// TIA Portal V18 program export: 1 tag tables, 1 data types, 57 data blocks, 50 code blocks (in call order from the OBs), 135 instance data blocks

VAR_GLOBAL   // PLC tag table "Default tag table"
   "Alarm Drive1" AT %I0.0 : Bool;
   "Alarm Drive 2" AT %I0.1 : Bool;
   setFlowRate AT %IW64 : Int;
   "AI on board(1)" AT %IW102 : Int;
   "preliminary empty signal component B1" AT %I0.6 : Bool;
   "Metering Start Foot Switch" AT %I1.2 : Bool;
   "Metering Start" AT %I1.3 : Bool;
   "Metering Stop" AT %I1.4 : Bool;
   "Metering Function Selection" AT %I2.0 : Bool;
   "Prerun Function" AT %I2.1 : Bool;
   "level empty signal component B1" AT %I0.7 : Bool;
   Flush AT %I2.2 : Bool;
   "Pressure sensor Pump Inlet A" AT %IW112 : Int;
   "Pressure Sensor Pump Inlet B" AT %IW114 : Int;
   "Pressure Sensor Pump Outlet A" AT %IW116 : Int;
   "Pressure Sensor Pump Outlet B" AT %IW118 : Int;
   "RPM PUMP A" AT %ID1008 : DInt;
   "RPM PUMP B" AT %ID1012 : DInt;
   "Level empty Signal component A1" AT %I0.3 : Bool;
   "program selection bit 3" AT %I2.6 : Bool;
   "preliminary empty signal component A1" AT %I0.2 : Bool;
   "Program selection bit0" AT %I2.3 : Bool;   //    {ExternalWritable false}
   "program selection bit 1" AT %I2.4 : Bool;
   "program selection bit2" AT %I2.5 : Bool;
   "Regenration Position Reached" AT %I1.5 : Bool;
   "reset pb" AT %I2.7 : Bool;
   "preliminary empty signal component A2" AT %I0.4 : Bool;
   "Level empty Signal component A2" AT %I0.5 : Bool;
   "preliminary empty signal component B2" AT %I1.0 : Bool;
   "level empty signal component B2" AT %I1.1 : Bool;
   "Level Sensor A" AT %IW120 : Int;
   "Level Sensor B" AT %IW122 : Int;
   "Pressure sensor Pump Inlet A_mA" AT %IW124 : Int;
   "Pressure Sensor Pump Inlet B_mA" AT %IW126 : Int;
   "emergency stop" AT %M3.5 : Bool;
   heater1 AT %IW144 : Int;
   heater2 AT %IW146 : Int;
   heater3 AT %IW148 : Int;
   heater4 AT %IW150 : Int;
   "Control ON" AT %I3.0 : Bool;
   "Control ON Led" AT %Q1.0 : Bool;
   "Reserve out3" AT %Q1.1 : Bool;
   "Metering Running" AT %Q2.2 : Bool;
   "ready to meter" AT %Q2.0 : Bool;
   "Metering Fault" AT %Q2.5 : Bool;
   "General Alarm" AT %Q2.1 : Bool;
   "Waiting for pre run" AT %Q2.3 : Bool;
   "metering Completed" AT %Q2.4 : Bool;
   "tower lamp yellow" AT %Q0.5 : Bool;
   "Reserve out0" AT %Q0.6 : Bool;
   "Reserve out1" AT %Q0.7 : Bool;
   "potlife error" AT %Q2.6 : Bool;
   "Reserve Output6" AT %Q2.7 : Bool;
   buzzer AT %Q0.4 : Bool;
   "Gear Pump A On_FWD" AT %Q0.0 : Bool;
   "Gear Pump B On_FWD" AT %Q0.2 : Bool;
   speedReference_ComponentB AT %QW130 : Int;
   speedReference_ComponentA AT %QW128 : Int;
   rampReference_ComponentA AT %QW132 : Int;
   rampReference_ComponentB AT %QW134 : Int;
   "Gear Pump A On_REW" AT %Q0.1 : Bool;
   "Gear Pump B On_REW" AT %Q0.3 : Bool;
   "Material 1 Temperature output" AT %Q3.0 : Bool;
   "Material 2 Temperature output" AT %Q3.1 : Bool;
   "Material 3 Temperature output" AT %Q3.2 : Bool;
   "Material 4 Temperature output" AT %Q3.3 : Bool;
   "gear Pump A fault" AT %M100.1 : Bool;
   "gear Pump B fault" AT %M100.2 : Bool;
   "Outlet Component A On" AT %M261.4 : Bool;
   "Outlet Component B On" AT %M200.4 : Bool;
   "program selection bit4" AT %M100.5 : Bool;
   "Agitator B Fault" AT %M100.3 : Bool;
   "Phase sequence relay Failure" AT %M100.4 : Bool;
   "Part Present sensor" AT %M100.0 : Bool;
   "Metering Ready" AT %M201.2 : Bool;
   "Tank A1 pressure" AT %MW240 : Int;
   "Tank A2 pressure" AT %MW242 : Int;
   "Tank B1 pressure" AT %MW244 : Int;
   "Tank Level A2" AT %MW248 : Int;
   "Gear Pump A Speed" AT %MW128 : Int;
   "Gear Pump B Speed" AT %MW130 : Int;
   "Mixer Speed" AT %MW208 : Int;
   "reserve  Analog output_0" AT %MW210 : Int;
   System_Byte AT %MB1 : Byte;
   FirstScan AT %M1.0 : Bool;
   DiagStatusUpdate AT %M1.1 : Bool;
   AlwaysTRUE AT %M1.2 : Bool;
   AlwaysFALSE AT %M1.3 : Bool;
   Clock_Byte AT %MB0 : Byte;
   Clock_10Hz AT %M0.0 : Bool;
   Clock_5Hz AT %M0.1 : Bool;
   "Clock_2.5Hz" AT %M0.2 : Bool;
   Clock_2Hz AT %M0.3 : Bool;
   "Clock_1.25Hz" AT %M0.4 : Bool;
   Clock_1Hz AT %M0.5 : Bool;
   "Clock_0.625Hz" AT %M0.6 : Bool;
   "Clock_0.5Hz" AT %M0.7 : Bool;
   "Fault register 1" AT %MW60 : Word;
   "Fault register 2" AT %MW62 : Word;
   "Fault register 3" AT %MW64 : Word;
   "Fault register 4" AT %MW66 : Word;
   "Fault register 5" AT %MW68 : Word;
   "A1-emergency stop active" AT %M61.0 : Bool;
   "A2-Pump A Drive Fault" AT %M61.1 : Bool;
   "A3-pump B drive Fault" AT %M61.2 : Bool;
   "A4-Agitator A1 fault" AT %M61.3 : Bool;
   "A5-Agitator A2 fault" AT %M61.4 : Bool;
   "A6-Tank A level sensor fault" AT %M61.5 : Bool;
   "A7-Tank B level sensor fault" AT %M61.6 : Bool;
   "A8-Pump A pressure sensor fault" AT %M61.7 : Bool;
   "A9-Pump B pressure sensor fault" AT %M60.0 : Bool;
   "A10-Tank A1 level sensor fault" AT %M60.1 : Bool;
   "A11-Tank A Filling Error" AT %M60.2 : Bool;
   "A12-Heater1 sensor fault" AT %M60.3 : Bool;
   "A13-Heater2 sensor fault" AT %M60.4 : Bool;
   "A14-Heater3 sensor fault" AT %M60.5 : Bool;
   "A15-Heater4 sensor fault" AT %M60.6 : Bool;
   "A16-Vaccum pump A fault" AT %M60.7 : Bool;
   "A17-Heater1 undertemperature" AT %M63.0 : Bool;
   "A18-Heater2 undertemperature" AT %M63.1 : Bool;
   "A19-Heater3 undertemperature" AT %M63.2 : Bool;
   "A20-Heater4 undertemperature" AT %M63.3 : Bool;
   "A21- Heater1 overtemperature" AT %M63.4 : Bool;
   "A22- Heater2 overtemperature" AT %M63.5 : Bool;
   "A23- Heater3 overtemperature" AT %M63.6 : Bool;
   "A24- Heater4 overtemperature" AT %M63.7 : Bool;
   "A25- Heater 8 pt100 discooneted" AT %M62.0 : Bool;
   "A26- Heater 9 pt100 discooneted" AT %M62.1 : Bool;
   "A27- Heater 10 pt100 discooneted" AT %M62.2 : Bool;
   "A28- Pump A over pressure" AT %M62.3 : Bool;
   "A29-pump B Over pressure" AT %M62.4 : Bool;
   "A30-Tank A1 Level Empty" AT %M62.5 : Bool;
   "A31-Tank A2 Level Empty" AT %M62.6 : Bool;
   "A32-Tank B Level Empty" AT %M62.7 : Bool;
   "A33-Tank A1 low level" AT %M65.0 : Bool;
   "A34-Tank A2 low level" AT %M65.1 : Bool;
   "A35-Tank B low level" AT %M65.2 : Bool;
   "A36-Pump A lower pressure" AT %M65.3 : Bool;
   "A37-Pump B lower pressure" AT %M65.4 : Bool;
   "A38-A material Supply fault" AT %M65.5 : Bool;
   "A39-B material Supply fault" AT %M65.6 : Bool;
   "A40-Potlife elapsed Change static mixer" AT %M65.7 : Bool;
   "A41- Heater 1 temperature Low" AT %M64.0 : Bool;
   "A42- Heater 2 temperature Low" AT %M64.1 : Bool;
   "A43- Heater 3 temperature Low" AT %M64.2 : Bool;
   "A44- Heater 4 temperature Low" AT %M64.3 : Bool;
   "A45- Heater 5 temperature Low" AT %M64.4 : Bool;
   "A46- Heater 6 temperature Low" AT %M64.5 : Bool;
   "A47- Heater 7 temperature Low" AT %M64.6 : Bool;
   "A48- Heater 8 temperature Low" AT %M64.7 : Bool;
   "A49- heater 9 temperature low" AT %M67.0 : Bool;
   "A50- heater 10 temperature low" AT %M67.1 : Bool;
   "A51- heater 1 temperature high" AT %M67.2 : Bool;
   "A52- heater 2 temperature high" AT %M67.3 : Bool;
   "A53- heater 3 temperature high" AT %M67.4 : Bool;
   "A54- heater 4 temperature high" AT %M67.5 : Bool;
   "A55- heater 5 temperature high" AT %M67.6 : Bool;
   "A56- heater 6 temperature high" AT %M67.7 : Bool;
   "A57- heater  7 temperature high" AT %M66.0 : Bool;
   "A58- heater 8 temperature high" AT %M66.1 : Bool;
   "A59- heater 9 temperature high" AT %M66.2 : Bool;
   "A60- heater 10 temperature high" AT %M66.3 : Bool;
   "A61- refilling failed Tank A1" AT %M66.4 : Bool;
   "A62-Error flowrate" AT %M66.5 : Bool;
   "A63- refilling failed Tank B" AT %M66.6 : Bool;
   Ack_A1 AT %M341.0 : Bool;
   Ack_A2 AT %M341.1 : Bool;
   Ack_A3 AT %M341.2 : Bool;
   Ack_A4 AT %M341.3 : Bool;
   Ack_A5 AT %M341.4 : Bool;
   Ack_A6 AT %M341.5 : Bool;
   Ack_A7 AT %M341.6 : Bool;
   Ack_A8 AT %M341.7 : Bool;
   Ack_A9 AT %M342.0 : Bool;
   Ack_A10 AT %M342.1 : Bool;
   Ack_A11 AT %M342.2 : Bool;
   Ack_A12 AT %M342.3 : Bool;
   Ack_A13 AT %M342.4 : Bool;
   Ack_A14 AT %M342.5 : Bool;
   Ack_A15 AT %M342.6 : Bool;
   Ack_A16 AT %M342.7 : Bool;
   Ack_A17 AT %M343.0 : Bool;
   Ack_A18 AT %M343.1 : Bool;
   Ack_A19 AT %M343.2 : Bool;
   Ack_A20 AT %M343.3 : Bool;
   Ack_A21 AT %M343.4 : Bool;
   Ack_A22 AT %M343.5 : Bool;
   Ack_A23 AT %M343.6 : Bool;
   Ack_A24 AT %M343.7 : Bool;
   Ack_A25 AT %M344.0 : Bool;
   Ack_A26 AT %M344.1 : Bool;
   Ack_A27 AT %M344.2 : Bool;
   Ack_A28 AT %M344.3 : Bool;
   Ack_A29 AT %M344.4 : Bool;
   Ack_A30 AT %M344.5 : Bool;
   Ack_A31 AT %M344.6 : Bool;
   Ack_A32 AT %M344.7 : Bool;
   Ack_A33 AT %M345.0 : Bool;
   Ack_A34 AT %M345.1 : Bool;
   Ack_A35 AT %M345.2 : Bool;
   Ack_A36 AT %M345.3 : Bool;
   Ack_A37 AT %M345.4 : Bool;
   Ack_A38 AT %M345.5 : Bool;
   Ack_A39 AT %M345.6 : Bool;
   Ack_A40 AT %M345.7 : Bool;
   Ack_A41 AT %M346.0 : Bool;
   Ack_A42 AT %M346.1 : Bool;
   Ack_A43 AT %M346.2 : Bool;
   Ack_A44 AT %M346.3 : Bool;
   Ack_A45 AT %M346.4 : Bool;
   Ack_A46 AT %M346.5 : Bool;
   Ack_A47 AT %M346.6 : Bool;
   Ack_A48 AT %M346.7 : Bool;
   Ack_A49 AT %M347.0 : Bool;
   Ack_A50 AT %M347.1 : Bool;
   Ack_A51 AT %M347.2 : Bool;
   Ack_A52 AT %M347.3 : Bool;
   Ack_A53 AT %M347.4 : Bool;
   Ack_A54 AT %M347.5 : Bool;
   Ack_A55 AT %M347.6 : Bool;
   Ack_A56 AT %M347.7 : Bool;
   Ack_A57 AT %M348.0 : Bool;
   Ack_A58 AT %M348.1 : Bool;
   Ack_A59 AT %M348.2 : Bool;
   Ack_A60 AT %M348.3 : Bool;
   Ack_A61 AT %M348.4 : Bool;
   Ack_A62 AT %M348.5 : Bool;
   Ack_A63 AT %M348.6 : Bool;
   Ack_A64 AT %M348.7 : Bool;
   Ack_A65 AT %M349.0 : Bool;
   Ack_A66 AT %M349.1 : Bool;
   Ack_A67 AT %M349.2 : Bool;
   Ack_A68 AT %M349.3 : Bool;
   Ack_A69 AT %M349.4 : Bool;
   Ack_hmi AT %M39.0 : Bool;
   Ack_site AT %M39.1 : Bool;
   Ack_PB AT %M39.2 : Bool;
   Fault_Ack_ONS AT %M39.3 : Bool;
   Tag_1 AT %M21.0 : Bool;
   Tag_2 AT %M4.1 : Bool;
   Ack_hmi_ons AT %M39.4 : Bool;
   "1sec_pulse" AT %M2.0 : Bool;
   "transperant backround" AT %M5.0 : Bool;
   "error count" AT %MD6 : UDInt;
   "A66-Tank A1 over pressure" AT %M69.1 : Bool;
   "A67-Tank A2 over pressure" AT %M69.2 : Bool;
   "A68-Tank B1 over pressure" AT %M69.3 : Bool;
   "Pgm No site" AT %MW23 : Int;
   "Pgm selection Bit memory 1" AT %M23.0 : Bool;
   "Pgm selection Bit memory 2" AT %M23.1 : Bool;
   "Pgm selection Bit memory 3" AT %M23.2 : Bool;
   "Pgm selection Bit memory 4" AT %M23.4 : Bool;
   "A69-mixer element break" AT %M69.4 : Bool;
   "Tank B2 pressure" AT %MW246 : Int;
   "Tank Level B2" AT %MW250 : Int;
   "VC1 new Pulse" AT %MD500 : DWord;
   "VC1 OLD Pulse" AT %MD504 : DWord;
   "VC2 new Pulse" AT %MD508 : DWord;
   "VC2 OLD Pulse" AT %MD512 : DWord;
   "VC1 Frequency" AT %MD516 : Real;
   "VC2 Frequency" AT %MD520 : Real;
   "VC1 Pulse in 1HZ" AT %MD524 : Real;
   "VC2 Pulse in 1HZ" AT %MD528 : Real;
   Tag_3 AT %MD1000 : DInt;
   Ack_A70 AT %M349.5 : Bool;
   Ack_A71 AT %M349.6 : Bool;
   Ack_A72 AT %M349.7 : Bool;
   Ack_A73 AT %M350.0 : Bool;
   "A70-mixing ratio low  warning" AT %M69.5 : Bool;
   "A71-mixing ratio high warning" AT %M69.6 : Bool;
   "A72-mixing ratio low fault" AT %M69.7 : Bool;
   "A89-Level Empty Drum B2" AT %M70.0 : Bool;
   "ready to power on servo" AT %M2.1 : Bool;
   "Pump Ready A1" AT %M100.6 : Bool;
   "Pump Ready A2" AT %M100.7 : Bool;
   "Pump Ready B1" AT %M101.0 : Bool;
   "Pump Ready B2" AT %M101.1 : Bool;
   Ack_A74 AT %M350.1 : Bool;
   Ack_A75 AT %M350.2 : Bool;
   Ack_A76 AT %M350.3 : Bool;
   Ack_A77 AT %M350.4 : Bool;
   Ack_A78 AT %M350.5 : Bool;
   Ack_A79 AT %M350.6 : Bool;
   Ack_A80 AT %M350.7 : Bool;
   Ack_A81 AT %M351.0 : Bool;
   Ack_A82 AT %M351.1 : Bool;
   Ack_A83 AT %M351.2 : Bool;
   Ack_A84 AT %M351.3 : Bool;
   Ack_A85 AT %M351.4 : Bool;
   Ack_A86 AT %M351.5 : Bool;
   Ack_A87 AT %M351.6 : Bool;
   Ack_A88 AT %M351.7 : Bool;
   Ack_A89 AT %M352.0 : Bool;
   Ack_A90 AT %M352.1 : Bool;
   Ack_A91 AT %M352.2 : Bool;
   Ack_A92 AT %M352.3 : Bool;
   Ack_A93 AT %M352.4 : Bool;
   Ack_A94 AT %M352.5 : Bool;
   Ack_A95 AT %M352.6 : Bool;
   Ack_A96 AT %M352.7 : Bool;
   Ack_A97 AT %M353.0 : Bool;
   Ack_A98 AT %M353.1 : Bool;
   Ack_A99 AT %M353.2 : Bool;
   Ack_A100 AT %M353.3 : Bool;
   Ack_A101 AT %M353.4 : Bool;
   Ack_A102 AT %M353.5 : Bool;
   Ack_A103 AT %M353.6 : Bool;
   Ack_A104 AT %M353.7 : Bool;
   Ack_A105 AT %M354.0 : Bool;
   Ack_A106 AT %M354.1 : Bool;
   Ack_A107 AT %M354.2 : Bool;
   Ack_A108 AT %M354.3 : Bool;
   Ack_A109 AT %M354.4 : Bool;
   Ack_A110 AT %M354.5 : Bool;
   Ack_A111 AT %M354.6 : Bool;
   Ack_A112 AT %M355.0 : Bool;
   Ack_A113 AT %M355.1 : Bool;
   Ack_A114 AT %M355.2 : Bool;
   Ack_A115 AT %M355.3 : Bool;
   Ack_A116 AT %M355.4 : Bool;
   Ack_A117 AT %M355.5 : Bool;
   Ack_A118 AT %M355.6 : Bool;
   Ack_A119 AT %M355.7 : Bool;
   Ack_A120 AT %M356.0 : Bool;
   Ack_A121 AT %M356.1 : Bool;
   Ack_A122 AT %M356.2 : Bool;
   Ack_A123 AT %M356.3 : Bool;
   Ack_A124 AT %M356.4 : Bool;
   Ack_A125 AT %M356.5 : Bool;
   Ack_A126 AT %M356.6 : Bool;
   Ack_A127 AT %M356.7 : Bool;
   Ack_A128 AT %M357.0 : Bool;
   Ack_A129 AT %M357.1 : Bool;
   Ack_A130 AT %M357.2 : Bool;
   Ack_A131 AT %M357.3 : Bool;
   Ack_A132 AT %M357.4 : Bool;
   Ack_A133 AT %M357.5 : Bool;
   Ack_A134 AT %M357.6 : Bool;
   Ack_A135 AT %M357.7 : Bool;
   Ack_A136 AT %M358.0 : Bool;
   Ack_A137 AT %M358.1 : Bool;
   Ack_A138 AT %M358.2 : Bool;
   Ack_A139 AT %M358.3 : Bool;
   Ack_A140 AT %M358.4 : Bool;
   Ack_A141 AT %M358.5 : Bool;
   Ack_A142 AT %M358.6 : Bool;
   Ack_A143 AT %M358.7 : Bool;
   "Fault register 6" AT %MW70 : Word;
   "Fault register 7" AT %MW72 : Word;
   "Fault register 8" AT %MW74 : Word;
   "Fault register 9" AT %MW76 : Word;
   Ack_A144 AT %M359.0 : Bool;
   Ack_A145 AT %M359.1 : Bool;
   Ack_A146 AT %M359.2 : Bool;
   Ack_A147 AT %M359.3 : Bool;
   Ack_A148 AT %M359.4 : Bool;
   Ack_A149 AT %M359.5 : Bool;
   Ack_A150 AT %M359.6 : Bool;
   Ack_A151 AT %M359.7 : Bool;
   Ack_A152 AT %M360.0 : Bool;
   Ack_A154 AT %M360.2 : Bool;
   Ack_A155 AT %M360.3 : Bool;
   Ack_A156 AT %M360.4 : Bool;
   Ack_A157 AT %M360.5 : Bool;
   Ack_A158 AT %M360.6 : Bool;
   Ack_A159 AT %M360.7 : Bool;
   Ack_A160 AT %M361.0 : Bool;
   "A82-Level Low Drum A1" AT %M71.1 : Bool;
   "A83-Level Low Drum B1" AT %M71.2 : Bool;
   "A84-Level Low Drum A2" AT %M71.3 : Bool;
   "A85-Level Low Drum B2" AT %M71.4 : Bool;
   "A86-Level Empty Drum A1" AT %M71.5 : Bool;
   "A87-Level Empty Drum B1" AT %M71.6 : Bool;
   "A88-Level Empty Drum A2" AT %M71.7 : Bool;
   Ack_A168 AT %M361.1 : Bool;
   Ack_A169 AT %M361.2 : Bool;
   Ack_A170 AT %M361.3 : Bool;
   Ack_A171 AT %M361.4 : Bool;
   Ack_A172 AT %M361.5 : Bool;
   Ack_A173 AT %M361.6 : Bool;
   Ack_A174 AT %M361.7 : Bool;
   Ack_A175 AT %M362.0 : Bool;
   Ack_A176 AT %M362.1 : Bool;
   Ack_A177 AT %M362.2 : Bool;
   Ack_A178 AT %M362.3 : Bool;
   Ack_A179 AT %M362.4 : Bool;
   Ack_A180 AT %M362.5 : Bool;
   Ack_A181 AT %M362.6 : Bool;
   Ack_A182 AT %M362.7 : Bool;
   Ack_A183 AT %M363.0 : Bool;
   Ack_A184 AT %M363.1 : Bool;
   Ack_A185 AT %M363.2 : Bool;
   Ack_A186 AT %M363.3 : Bool;
   Ack_A187 AT %M363.4 : Bool;
   Ack_A188 AT %M363.5 : Bool;
   "Fault register 10" AT %MW32 : Word;
   "A74-Level Low Pressure Vessel A" AT %M68.1 : Bool;
   "A75-Level Low Pressure Vessel B" AT %M68.2 : Bool;
   "A76-Level Empty Pressure Vessel A" AT %M68.3 : Bool;
   "A77-Level Empty Pressure Vessel B" AT %M68.4 : Bool;
   "A78-Level Low Catridge A" AT %M68.5 : Bool;
   "A79-Level Low Catridge B" AT %M68.6 : Bool;
   "A80-Level Empty Catridge A" AT %M68.7 : Bool;
   Tag_4 AT %M73.0 : Bool;
   Tag_5 AT %M73.1 : Bool;
   Tag_6 AT %M73.2 : Bool;
   Tag_7 AT %M73.3 : Bool;
   Tag_8 AT %M73.4 : Bool;
   Tag_9 AT %M73.5 : Bool;
   Tag_10 AT %M73.6 : Bool;
   Tag_11 AT %M73.7 : Bool;
   "A90 Pressure sensor Pump A Outlet Fault" AT %M72.0 : Bool;
   "A91 Pressure sensor Pump B Outlet Fault" AT %M72.1 : Bool;
   "A92 Over pressure A outlet" AT %M72.2 : Bool;
   "A93 Over pressure B outlet" AT %M72.3 : Bool;
   "A94- Pump A Outlet Under Pressure" AT %M72.4 : Bool;
   "A95- Pump B Outlet Under Pressure" AT %M72.5 : Bool;
   Tag_18 AT %M72.6 : Bool;
   Tag_19 AT %M72.7 : Bool;
   Tag_20 AT %M75.0 : Bool;
   Tag_21 AT %M75.1 : Bool;
   Tag_22 AT %M75.2 : Bool;
   Tag_23 AT %M75.3 : Bool;
   Tag_24 AT %M75.4 : Bool;
   Tag_25 AT %M75.5 : Bool;
   Tag_26 AT %M75.6 : Bool;
   Tag_27 AT %M75.7 : Bool;
   Tag_28 AT %M74.0 : Bool;
   Tag_29 AT %M74.1 : Bool;
   Tag_30 AT %M74.2 : Bool;
   Tag_31 AT %M74.3 : Bool;
   Tag_32 AT %M74.4 : Bool;
   Tag_33 AT %M74.5 : Bool;
   Tag_34 AT %M74.6 : Bool;
   Tag_35 AT %M74.7 : Bool;
   Tag_36 AT %M77.0 : Bool;
   Tag_37 AT %M77.1 : Bool;
   Tag_38 AT %M77.2 : Bool;
   Tag_39 AT %M77.3 : Bool;
   Tag_40 AT %M77.4 : Bool;
   Tag_41 AT %M77.5 : Bool;
   Tag_42 AT %M77.6 : Bool;
   Tag_43 AT %M77.7 : Bool;
   Tag_44 AT %M76.0 : Bool;
   Tag_45 AT %M76.1 : Bool;
   Tag_46 AT %M76.2 : Bool;
   Tag_47 AT %M76.3 : Bool;
   Tag_48 AT %M76.4 : Bool;
   Tag_49 AT %M76.5 : Bool;
   Tag_50 AT %M76.6 : Bool;
   Tag_51 AT %M76.7 : Bool;
   Ack_A153 AT %M360.1 : Bool;
   "Inlet Component A On" AT %M261.2 : Bool;
   "Inlet Component B On" AT %M261.3 : Bool;
   "Agitator B" AT %M200.3 : Bool;
   "Material refilling A" AT %M200.5 : Bool;
   "Material refilling B" AT %M200.6 : Bool;
   "Refilling Pump A" AT %M200.7 : Bool;
   "Refilling Pump B" AT %M201.0 : Bool;
   "Reserve Output 3" AT %M201.1 : Bool;
   "Pressure Release A" AT %M200.2 : Bool;
   "Pressure Release B" AT %M201.3 : Bool;
   "A64- No siganl RPM sensor A" AT %M70.2 : Bool;
   "A65- No siganl RPM sensor B" AT %M70.3 : Bool;
   "A70-Warning mixing ratio low" AT %M70.4 : Bool;
   "A71- warning Mixing Ratio high" AT %M70.5 : Bool;
   "A72- Error Mixing ratio Low" AT %M70.6 : Bool;
   "A73- Error Mixing Ratio high" AT %M70.7 : Bool;
   Tag_52 AT %M30.0 : Bool;
   Tag_53 AT %M30.1 : Bool;
   Tag_54 AT %M500.0 : Bool;
   tnp AT %M2.2 : Bool;
   "PID A setpoint scaled" AT %MD10 : Real;
   "PID A input scaled" AT %MD14 : Real;
   "PID B setpoint scaled" AT %MD34 : Real;
   "PID B input scaled" AT %MD40 : Real;
   dummy1 AT %M2.3 : Bool;
   "RTD OUTPUT" AT %MD44 : Real;
   "RTD OUTPUT1" AT %MD48 : Real;
   "prg no sel" AT %MW18 : Int;
   "SD Logg" AT %MD52 : UDInt;
   "SD LOG TRIGGER" AT %M2.5 : Bool;
   "USB Logg" AT %MD140 : UDInt;
   "USB LOG TRIGGER" AT %M2.6 : Bool;
   "A81-Level Empty Catridge B" AT %M71.0 : Bool;
   TempPE1 AT %M2.7 : Bool;
   TempPE2 AT %M3.0 : Bool;
   temps AT %MD102 : Real;
   temp_unitsel AT %MW56 : Int;
   test AT %M3.1 : Bool;
   snuffback_completed AT %M3.2 : Bool;
   temp_dispese_qty AT %MD26 : Real;
   RatioCheck_status AT %MW78 : Int;
   actual_gramA_Old AT %MD106 : Real;
   actual_gramB_Old AT %MD110 : Real;
   Function_snuffback_selected AT %M3.3 : Bool;
   start_snuffback AT %M3.4 : Bool;
   "Fault display register 1" AT %MW80 : Word;
   "Fault display register 2" AT %MW82 : Word;
   "Fault display register 3" AT %MW84 : Word;
   "Fault display register 4" AT %MW86 : Word;
   "Fault display register 5" AT %MW88 : Word;
   "Fault display register 6" AT %MW90 : Word;
   "Fault display register 7" AT %MW92 : Word;
   machine_on AT %M2.4 : Bool;
   estop AT %I3.1 : Bool;
END_VAR

TYPE "Condition_Check"
// stored: IsFailsafeCompliant false
   STRUCT
      Date_time : DTL;
      Pressure_achieve_time : DInt;
      Leakage_Pressure : Real;
      Status : Int;
   END_STRUCT;
END_TYPE

DATA_BLOCK "Agitator"   // DB124
{ S7_Optimized_Access := 'TRUE' }
VERSION : 0.1
// stored: AutoNumber true, DBAccessibleFromOPCUA true, IsOnlyStoredInLoadMemory false, IsRetainMemResEnabled false, IsWriteProtectedInAS false, MemoryReserve 100
   VAR
      Control : Struct
         A1 : Struct
            "Show ON Button" : Bool;
            "Show OFF Button" : Bool;
            ON : Bool;
            OFF : Bool;
            "ON timer okay" : Bool;
            "Off timer Okay" : Bool;
            "Off hmi" : Bool;
            selected : Bool;
            Run : Bool;
            "ON hmi" : Bool;
         END_STRUCT;
         A2 : Struct
            ON : Bool;
            OFF : Bool;
            "ON hmi" : Bool;
            "ON timer okay" : Bool;
            "Off timer Okay" : Bool;
            selected : Bool;
            "Off hmi" : Bool;
            Run : Bool;
            "Show ON Button" : Bool;
            "Show OFF Button" : Bool;
         END_STRUCT;
         B1 : Struct
            ON : Bool;
            "ON hmi" : Bool;
            OFF : Bool;
            "ON timer okay" : Bool;
            "Off timer Okay" : Bool;
            selected : Bool;
            "Off hmi" : Bool;
            Run : Bool;
            "Show ON Button" : Bool;
            "Show OFF Button" : Bool;
         END_STRUCT;
      END_STRUCT;
   END_VAR
   VAR RETAIN
      "Time" : Struct
         A1 : Struct
            "ON time" : Int;
            "OFF time" : Int;
         END_STRUCT;
         A2 : Struct
            "ON time" : Int;
            "OFF time" : Int;
         END_STRUCT;
         B1 : Struct
            "ON time" : Int;
            "OFF time" : Int;
         END_STRUCT;
      END_STRUCT;
      selection : Struct
         A1 : Int;
         A2 : Int;
         B1 : Int;
      END_STRUCT;
   END_VAR
   VAR
      "Time control" : Struct
         A1 : Struct
            "ON time" : Time;
            "OFF time" : Time;
         END_STRUCT;
         A2 : Struct
            "ON time" : Time;
            "OFF time" : Time;
         END_STRUCT;
         B1 : Struct
            "ON time" : Time;
            "OFF time" : Time;
         END_STRUCT;
      END_STRUCT;
      "ON HMI" : Bool;
      "Display ON Button" : Bool;
      "Display Off Button" : Bool;
      "Run time PV" : Struct
         A1 : Int;
         A2 : Int;
         B1 : Int;
      END_STRUCT;
      "Idle time PV" : Struct
         A1 : Int;
         A2 : Int;
         B1 : Int;
      END_STRUCT;
      "Run time PVms" : Struct
         A1 : DInt;
         A2 : DInt;
         B1 : DInt;
      END_STRUCT;
      "Idle time PVmS" : Struct
         A1 : DInt;
         A2 : DInt;
         B1 : DInt;
      END_STRUCT;
   END_VAR
BEGIN
END_DATA_BLOCK

DATA_BLOCK "Control"   // DB68
{ S7_Optimized_Access := 'TRUE' }
VERSION : 0.1
// stored: AutoNumber true, DBAccessibleFromOPCUA true, IsOnlyStoredInLoadMemory false, IsRetainMemResEnabled false, IsWriteProtectedInAS false, MemoryReserve 100
   VAR
      "waiting For pre run" : Bool := TRUE;
      "ready for operation" : Bool := FALSE;
      "metering blocked" : Bool := FALSE;
      "change Screen" : Int := 0;
      "A metering ready" : Bool := TRUE;
      "B metering ready" : Bool := TRUE;
      "A&B metering ready" : Bool := TRUE;
      "metering program ready" : Bool := FALSE;
      "Evacuation Ready Tank A1" : Bool := FALSE;
      "Evacuation Ready Tank A2" : Bool := FALSE;
      "Evacuation Read" : Bool := FALSE;
      "Recirculation Enabled" : Bool := FALSE;
      "recirculation okay" : Bool := FALSE;
      "Show start Button" : Bool := FALSE;
      "Show esc Button" : Bool := FALSE;
      "Show stop Button" : Bool := FALSE;
      "Do not show para& config button" : Bool := FALSE;
   END_VAR
   VAR RETAIN
      "Start signal on site type" : Int := 1;
      "stop signal on site type" : Int := 0;
      "Program selection Mode" : Int := 0;
      "Flowrate adjustment type" : Int := 0;
   END_VAR
   VAR
      "A recirculation Ready" : Bool := FALSE;
      "B recirculation Ready" : Bool := FALSE;
      "recirculation ready" : Bool := FALSE;
      "Show alarm field" : Bool := FALSE;
      "Flush ready" : Bool := TRUE;
      "ratio check Ready" : Bool := TRUE;
      "reset from hmi _site_pb_PN" : Bool := FALSE;
      "start from hmi_site_pb_PN" : Bool := FALSE;
      "stop from hmi_site_pb_PN" : Bool := FALSE;
      "Heater OK" : Bool := FALSE;
      "Heater No Fault" : Bool := FALSE;
   END_VAR
   VAR RETAIN
      "Pump A maximum Idle Time" : Int := 30;
      "Pump B maximum Idle Time" : Int := 30;
   END_VAR
   VAR
      "Pump A maximum Idle Time sec" : DInt := 1800000;
      "Pump B maximum Idle Time sec" : DInt := 1800000;
      Mute : Struct
         "Mute enable" : Bool := FALSE;
         "Mute buzzer" : Bool := FALSE;
         "Mutte On" : Bool := FALSE;
      END_STRUCT;
      Pressure_sensor_select : Int := 0;
   END_VAR
   VAR RETAIN
      Level_sensor_enable : Bool := FALSE;
      "Minimum Dispesing qty" : Real;
      "Minimum Snuff back qty" : Real;
      "Outlet On_off" : Bool;
   END_VAR
   VAR
      "Outlet On_off_disp" : Bool;
   END_VAR
BEGIN
END_DATA_BLOCK

DATA_BLOCK "DB_Recipe"   // DB290
{ S7_Optimized_Access := 'TRUE' }
VERSION : 0.1
// stored: AutoNumber true, DBAccessibleFromOPCUA true, IsOnlyStoredInLoadMemory false, IsRetainMemResEnabled false, IsWriteProtectedInAS false, MemoryReserve 100
   VAR
      HMI_Recipe : Int := 0;
      HMI_Recipe_Data : String := '';
      Recepie_name : String;
   END_VAR
BEGIN
END_DATA_BLOCK

DATA_BLOCK "Data_block_1"   // DB26
{ S7_Optimized_Access := 'TRUE' }
VERSION : 0.1
// stored: AutoNumber true, DBAccessibleFromOPCUA true, IsOnlyStoredInLoadMemory false, IsRetainMemResEnabled false, IsWriteProtectedInAS false, MemoryReserve 100
   VAR
      on : Bool;
      outmin : Int;
      outhout : Int;
   END_VAR
BEGIN
END_DATA_BLOCK

DATA_BLOCK "DataloggingDB"   // DB98
{ S7_Optimized_Access := 'FALSE' }
VERSION : 0.1
// stored: AutoNumber true, DBAccessibleFromOPCUA true, IsOnlyStoredInLoadMemory false, IsWriteProtectedInAS false
   VAR RETAIN
      Enable : Bool := false;
      "TXt/csv" : Bool := false;
      "Sdcard/pendrive" : Int := 0;
      "trigger SD card logging" : Bool := false;
      "trigger pendrive logging" : Bool := false;
      Data : Struct
         "Date" : DTL := DTL#1970-01-01-00:00:00;
         "Time" : Time_Of_Day := TOD#00:00:00;
         "Blade Number" : String := '';
         operator : Int := 0;
         "Batch A" : String[25] := '';
         "Batch B" : String[25] := '';
         IDVCA : String[25] := '';
         IDVCB : String[25] := '';
         "Pressure outlet A" : Real := 0.0;
         "Pressure outlet B" : Real := 0.0;
         "Ratio Control Size" : Real := 0.0;
         "Ratio A100:B" : Real := 0.0;
         "Ratio Min" : Real := 0.0;
         "Ratio Max" : Real := 0.0;
         CPK : Real := 0.0;
         "Event Number" : UDInt := 0;
         Function : String[25] := '';
         Error : UDInt := 0;
         "Temp.inlet Heater A" : Real := 0.0;
         "Temp.At mixing  Block A" : Real := 0.0;
         "Temp.At mixing Block B" : Real := 0.0;
         "Temp.At Resin outlet" : Real := 0.0;
      END_STRUCT;
      "Data string" : Struct
         "Pressure outlet A" : String[25] := '';
         "Pressure outlet B" : String[25] := '';
         "Ratio Control Size" : String[25] := '';
         "Ratio A100:B" : String[25] := '';
         "Ratio Min" : String[25] := '';
         "Ratio Max" : String[25] := '';
         CPK : String[25] := '';
         Function : String[25] := '';
         "Temp.inlet Heater A" : String[25] := '';
         "Temp.At mixing  Block A" : String[25] := '';
         "Temp.At mixing Block B" : String[25] := '';
         "Temp.At Resin outlet" : String[25] := '';
         "Total A flush" : String[25] := '';
         "Total B flush" : String[25] := '';
         "Total Size" : String[25] := '';
         "metering Size" : String[25] := '';
         "Shot Size A" : String[25] := '';
         "Shot Size B" : String[25] := '';
         "Total Size A" : String[25] := '';
         "Total Size B" : String[25] := '';
      END_STRUCT;
      Data_1 : Struct
         "Total A flush" : Real := 0.0;
         "Total B flush" : Real := 0.0;
         "Total Size" : Real := 0.0;
         "metering Size" : Real := 0.0;
         "Total size A" : Real := 0.0;
         "Total size B" : Real := 0.0;
         "MOULD NOMINAL PRESSURE" : Real := 0.0;
      END_STRUCT;
      "Copy Flush A qty" : Bool := false;
      "Copy Dearate A Qty" : Bool := false;
      "Copy Flush B qty" : Bool := false;
      "Copy Dearate B Qty" : Bool := false;
      "Copy Ab Qty" : Bool := false;
      "Total Size calculation" : Struct
         "Previous value" : Real := 0.0;
         "volume dispensed" : Real := 0.0;
         "present value" : Real := 0.0;
         "Value to add" : Real := 0.0;
         "start copy" : Bool := false;
         "dosing running" : Bool := false;
      END_STRUCT;
      "Total Size A calculation" : Struct
         "Previous value" : Real := 0.0;
         "volume dispensed" : Real := 0.0;
         "present value" : Real := 0.0;
         "Value to add" : Real := 0.0;
         "start copy" : Bool := false;
         "dosing running" : Bool := false;
      END_STRUCT;
      "Total Size B calculation" : Struct
         "Previous value" : Real := 0.0;
         "volume dispensed" : Real := 0.0;
         "present value" : Real := 0.0;
         "Value to add" : Real := 0.0;
         "start copy" : Bool := false;
         "dosing running" : Bool := false;
      END_STRUCT;
      "Ready to Log" : Bool := false;
      "Log Done" : Bool := false;
      "No.of counts to calculate CPK" : Int := 0;
      "reset A flush" : Bool := false;
      "reset B flush" : Bool := false;
      "reset total Size" : Bool := false;
      "Process Data Start/Stop" : Real := 0.0;
      "30sec timer done" : Bool := false;
      datacollection : Struct
         day : String[4] := '';
         month : String[4] := '';
         year : String[6] := '';
         filename : String[15] := 'Dopag_';
      END_STRUCT;
      date_time : DTL;
      current_day : UDInt;
      previous_day : UDInt;
      current_week : UDInt;
      previous_week : UDInt;
      current_month : UDInt;
      previous_month : UDInt;
      day_changed : Bool;
      week_changed : Bool;
      month_changed : Bool;
      totalsizepreviousday : Real;
      totalsizeday : Real;
      totalsizeweek : Real;
      totalsizepreviousweek : Real;
      totalsizemonth : Real;
      totalsizepreviousmonth : Real;
      Total_Production_metering : Real;
      Total_Production_Prerun : Real;
      Total_Production_Ratiocheck : Real;
      Total_Production_regeneration : Real;
      Total_Production_Flush : Real;
      Total_Volume : Real;
      Reset_total_volume : Bool;
      "Metering%" : Real;
      "Prerun%" : Real;
      "Ratiocheck%" : Real;
      "Regen%" : Real;
      "Flush%" : Real;
      "Last reset" : DTL;
   END_VAR
BEGIN
END_DATA_BLOCK

DATA_BLOCK "Faults&warnings"   // DB67
{ S7_Optimized_Access := 'TRUE' }
VERSION : 0.1
// stored: AutoNumber true, DBAccessibleFromOPCUA true, IsOnlyStoredInLoadMemory false, IsRetainMemResEnabled false, IsWriteProtectedInAS false, MemoryReserve 100
   VAR
      "Critical Alarm Metering A" : Bool;
      "Critical Alarm metering B" : Bool;
      "Critical Alarm metering A&B" : Bool;
      "alarm Level" : Int;
      "Alarm popped" : Bool;
      "Alarm Number" : Int;
      "Alarm ack Hmi" : Bool;
      "Alarm class" : Int;
      "Fault display register" : Int;
      "Fault display register Moved" : Int;
      "Fault present" : Bool;
      "Status Nok" : Struct
         "Drive controller A NK" : Bool;
         "Drive controller B NK" : Bool;
         "Agitator A Fault" : Bool;
         "Agitator B Fault" : Bool;
         "Mixer Drive NK" : Bool;
         "Pressure sensor Pump A Inlet" : Bool;
         "Pressure Sensor Pump B Inlet" : Bool;
         "Pressure sensor Pump A Outlet" : Bool;
         "Pressure Sensor Pump B Outlet" : Bool;
         "Over pressure A inlet" : Bool;
         "Over pressure B inlet" : Bool;
         "Over pressure A outlet" : Bool;
         "Over pressure B outlet" : Bool;
         "Emergency stop" : Bool;
         "Control ON" : Bool;
         "Pressure sensor vessel A1" : Bool;
         "Pressure sensor vessel A2" : Bool;
         "Pressure sensor vessel B1" : Bool;
         "Pressure sensor vessel B2" : Bool;
         "Material Supply A" : Bool;
         "Material Supply B" : Bool;
         "Low level B2" : Bool;
         "Level Empty B2" : Bool;
         "Level sensor B2" : Bool;
         "Low level A1" : Bool;
         "Level empty A1" : Bool;
         "Level Sensor Pressure vessel A" : Bool;
         "Low level A2" : Bool;
         "Level empty A2" : Bool;
         "Low level B1" : Bool;
         "Level empty B1" : Bool;
         "Level Sensor Pressure vessel B" : Bool;
         "Flowrate error" : Bool;
         "Level Low Pressure Vessel A" : Bool;
         "Level Low Pressure Vessel B" : Bool;
         "Level Empty Pressure Vessel A" : Bool;
         "Level Empty Pressure Vessel B" : Bool;
         "Level Low Catridge A" : Bool;
         "Level Low Catridge B" : Bool;
         "Level Empty Catridge A" : Bool;
         "Level Empty Catridge B" : Bool;
         "Level Low Drum A1" : Bool;
         "Level Low Drum B1" : Bool;
         "Level Low Drum A2" : Bool;
         "Level Low Drum B2" : Bool;
         "Level Empty Drum A1" : Bool;
         "Level Empty Drum B1" : Bool;
         "Level Empty Drum A2" : Bool;
         "Level Empty Drum B2" : Bool;
      END_STRUCT;
      "Operator message 1" : Int;
      "Operator message 2" : Int;
      "alarm popped out" : Bool;
      "faultnumber in hmi" : Int;
      "alarm Display number" : Int;
      "Current Scroll Number" : DInt := 1;
   END_VAR
BEGIN
END_DATA_BLOCK

DATA_BLOCK "Flowrate adjustment A"   // DB78
{ S7_Optimized_Access := 'TRUE' }
VERSION : 0.1
// stored: AutoNumber true, DBAccessibleFromOPCUA true, IsOnlyStoredInLoadMemory false, IsRetainMemResEnabled false, IsWriteProtectedInAS false, MemoryReserve 100
   VAR RETAIN
      percentage : Struct
         "5%" : Real;
         "10%" : Real;
         "15%" : Real;
         "20%" : Real;
         "25%" : Real;
         "30%" : Real;
         "40%" : Real;
         "50%" : Real;
         "60%" : Real;
         "70%" : Real;
         "80%" : Real;
         "90%" : Real;
         "100%" : Real;
      END_STRUCT;
   END_VAR
   VAR
      "Reset Flowadjustment A" : Bool;
   END_VAR
BEGIN
END_DATA_BLOCK

DATA_BLOCK "Flowrate adjustment B"   // DB79
{ S7_Optimized_Access := 'TRUE' }
VERSION : 0.1
// stored: AutoNumber false, DBAccessibleFromOPCUA true, IsOnlyStoredInLoadMemory false, IsRetainMemResEnabled false, IsWriteProtectedInAS false, MemoryReserve 100
   VAR RETAIN
      percentage : Struct
         "5%" : Real;
         "10%" : Real;
         "15%" : Real;
         "20%" : Real;
         "25%" : Real;
         "30%" : Real;
         "40%" : Real;
         "50%" : Real;
         "60%" : Real;
         "70%" : Real;
         "80%" : Real;
         "90%" : Real;
         "100%" : Real;
      END_STRUCT;
   END_VAR
   VAR
      "Reset Flowadjustment B" : Bool;
   END_VAR
BEGIN
END_DATA_BLOCK

DATA_BLOCK "Flowrate"   // DB205
{ S7_Optimized_Access := 'TRUE' }
VERSION : 0.1
// stored: AutoNumber true, DBAccessibleFromOPCUA true, IsOnlyStoredInLoadMemory false, IsRetainMemResEnabled false, IsWriteProtectedInAS false, MemoryReserve 100
   VAR
      Current : Struct
         "A" : Real;
         "B" : Real;
         Mixed : Real;
      END_STRUCT;
      "current in ml/min" : Struct
         "A" : Real;
         "B" : Real;
         Mixed : Real;
      END_STRUCT;
      "current in L/min" : Struct
         "A" : Real;
         "B" : Real;
         Mixed : Real;
      END_STRUCT;
      "current in KG/min" : Struct
         "A" : Real;
         "B" : Real;
         Mixed : Real;
      END_STRUCT;
      "Volume in ml" : Struct
         "A" : Real;
         "B" : Real;
         mixed : Real;
      END_STRUCT;
      "Volume in L" : Struct
         "A" : Real;
         "B" : Real;
         mixed : Real;
      END_STRUCT;
      "Volume in Kg" : Struct
         "A" : Real;
         "B" : Real;
         mixed : Real;
      END_STRUCT;
      "Current Volume" : Struct
         "A" : Real;
         "B" : Real;
         mixed : Real;
      END_STRUCT;
      "Current Flowrate" : Struct
         "A" : Real;
         "B" : Real;
         mixed : Real;
      END_STRUCT;
   END_VAR
   VAR RETAIN
      "selection ml/lit/kg" : Int := 1;
   END_VAR
   VAR
      Selected : Struct
         ml : Bool;
         cm3 : Bool;
         litre : Bool;
         kg : Bool;
         g { ExternalAccessible := 'False'; ExternalVisible := 'False'; ExternalWritable := 'False'} : Bool;
      END_STRUCT;
      tolerence : Struct
         Mixed : Real;
         Percentage : Real;
         "Mixed +" : Real;
         "Mixed -" : Real;
         Error : Bool;
      END_STRUCT;
      "current in g/min" : Struct
         "A" : Real;
         "B" : Real;
         Mixed : Real;
      END_STRUCT;
      "Volume in g" : Struct
         "A" : Real;
         "B" : Real;
         mixed : Real;
      END_STRUCT;
   END_VAR
BEGIN
END_DATA_BLOCK

DATA_BLOCK "Function ConditionCheck without valve"   // DB135
{ S7_Optimized_Access := 'TRUE' }
VERSION : 0.1
// stored: AutoNumber true, DBAccessibleFromOPCUA true, IsOnlyStoredInLoadMemory false, IsRetainMemResEnabled false, IsWriteProtectedInAS false, MemoryReserve 100
   VAR
      "Control A" : Struct
         "start Condition Check" : Bool := FALSE;
         "Condition Check running" : Bool := FALSE;
         "stop Condition Check" : Bool := FALSE;
         "Condition Check Completed" : Bool := FALSE;
         "Pressure Setpoint" : Real := 0.0;
         Check_Time : DInt := 0;
         Pressure_tolerance : Real := 0.0;
         "Time tolerance" : Real := 0.0;
         "installtaion mode" : Bool := TRUE;
      END_STRUCT;
      "Control B" : Struct
         "start Condition Check" : Bool := FALSE;
         "Condition Check running" : Bool := FALSE;
         "stop Condition Check" : Bool := FALSE;
         "Condition Check Completed" : Bool := FALSE;
         "Pressure Setpoint" : Real := 0.0;
         Check_Time : DInt := 0;
         Pressure_tolerance : Real := 0.0;
         "Time tolerance" : Real := 0.0;
         "installation mode" : Bool := TRUE;
      END_STRUCT;
      "Output A" : Struct
         "ON pump" : Bool := FALSE;
         "running time" : Int := 0;
         "ON_inlet A" : Bool := FALSE;
         Pressure_OK : Bool := FALSE;
         Pressure_NOK : Bool := FALSE;
         Pressure_release_time : DInt := 0;
         Test_Fail : Bool := FALSE;
         "Test Pass" : Bool := FALSE;
      END_STRUCT;
      "Output B" : Struct
         "ON pump" : Bool := FALSE;
         "running time" : Int := 0;
         "ON_inlet B" : Bool := FALSE;
         Pressure_OK : Bool := FALSE;
         Pressure_NOK : Bool := FALSE;
         Pressure_release_time : DInt := 15;
         Test_Fail : Bool := FALSE;
         "Test Pass" : Bool := FALSE;
      END_STRUCT;
   END_VAR
   VAR RETAIN
      "Input A" : Struct
         "set time" : Int := 20;
         "set flowrate" : Real := 5.0;
         "Pressure Setpoint" : Real := 10.0;
         Check_Time : DInt := 15;
         Pressure_tolerance : Real := 3.0;
         PressurisingSP : Real := 5.0;
         Pressurisingtime : DInt := 45;
      END_STRUCT;
      "Input B" : Struct
         "set time" : Int := 20;
         "set flowrate" : Real := 5.0;
         "Pressure Setpoint" : Real := 10.0;
         Check_Time : DInt := 15;
         Pressure_tolerance : Real := 3.0;
         PressurisingSP : Real := 5.0;
         Pressurisingtime : DInt := 45;
      END_STRUCT;
   END_VAR
   VAR
      "start time" : DTL := DTL#1970-01-01-00:00:00;
      Stoptime : DTL := DTL#1970-01-01-00:00:00;
      "time in ms" : DInt := 0;
   END_VAR
   VAR RETAIN
      "Data A" : Struct
         "Pressure Achieved time @installation" : DInt := 92;
         "Pressure time @operation" : DInt := 0;
         "Pressure Achieved time @ operation" : Array[0..20] of DInt;
         "Leakage test pressure" : Real := 0.0;
         Test_Data : Array[1..20] of "Condition_Check";
         temp_Test_Data { S7_SetPoint := 'True'} : "Condition_Check";
      END_STRUCT;
      "Data B" : Struct
         "Pressure Achieved time @installation" : DInt := 71;
         "Pressure time @operation" : DInt := 0;
         "Pressure Achieved time @ operation" : Array[0..20] of DInt;
         "Leakage test pressure" : Real := 0.0;
         Test_Data : Array[1..20] of "Condition_Check";
         temp_Test_Data { S7_SetPoint := 'True'} : "Condition_Check";
      END_STRUCT;
   END_VAR
   VAR
      reset_FIFOA { S7_SetPoint := 'True'} : Bool := FALSE;
      reset_FIFOB : Bool := FALSE;
      Show_popupA : Bool := FALSE;
      Show_popupB : Bool := FALSE;
   END_VAR
   VAR RETAIN
      Condition_check_en : Bool := TRUE;
   END_VAR
   VAR
      start_revA_condcheck : Bool := FALSE;
      RevA_time : DInt := 3000;
   END_VAR
   VAR RETAIN
      RevA_flowrate : Real := 1.0;
   END_VAR
   VAR
      start_revB_condcheck : Bool := FALSE;
      RevB_time : DInt := 3000;
   END_VAR
   VAR RETAIN
      RevB_flowrate : Real := 1.0;
   END_VAR
BEGIN
   "Data A"."Pressure Achieved time @ operation"[0..20] := 0;
   "Data A".Test_Data[1].Date_time := DTL#2012-01-05-00:30:04.579546;
   "Data A".Test_Data[2].Date_time := DTL#2012-01-05-00:39:31.124577;
   "Data A".Test_Data[3..20].Date_time := DTL#1970-01-01-00:00:00;
   "Data A".Test_Data[1..2].Pressure_achieve_time := 92;
   "Data A".Test_Data[3..20].Pressure_achieve_time := 0;
   "Data A".Test_Data[1].Leakage_Pressure := 6.67;
   "Data A".Test_Data[2..20].Leakage_Pressure := 0.0;
   "Data A".Test_Data[1..2].Status := 2;
   "Data A".Test_Data[3..20].Status := 0;
   "Data A".temp_Test_Data.Date_time := DTL#1970-01-01-00:00:00;
   "Data A".temp_Test_Data.Pressure_achieve_time := 0;
   "Data A".temp_Test_Data.Leakage_Pressure := 0.0;
   "Data A".temp_Test_Data.Status := 0;
   "Data B"."Pressure Achieved time @ operation"[0..20] := 0;
   "Data B".Test_Data[1].Date_time := DTL#2012-01-05-00:42:23.319592;
   "Data B".Test_Data[2].Date_time := DTL#2012-01-05-00:50:51.810518;
   "Data B".Test_Data[3..20].Date_time := DTL#1970-01-01-00:00:00;
   "Data B".Test_Data[1].Pressure_achieve_time := 26;
   "Data B".Test_Data[2].Pressure_achieve_time := 71;
   "Data B".Test_Data[3..20].Pressure_achieve_time := 0;
   "Data B".Test_Data[1].Leakage_Pressure := 14.28;
   "Data B".Test_Data[2].Leakage_Pressure := 11.56;
   "Data B".Test_Data[3..20].Leakage_Pressure := 0.0;
   "Data B".Test_Data[1].Status := 2;
   "Data B".Test_Data[2].Status := 1;
   "Data B".Test_Data[3..20].Status := 0;
   "Data B".temp_Test_Data.Date_time := DTL#1970-01-01-00:00:00;
   "Data B".temp_Test_Data.Pressure_achieve_time := 0;
   "Data B".temp_Test_Data.Leakage_Pressure := 0.0;
   "Data B".temp_Test_Data.Status := 0;
END_DATA_BLOCK

DATA_BLOCK "Function Continous Metering pgm"   // DB49
{ S7_Optimized_Access := 'TRUE' }
VERSION : 0.1
// stored: AutoNumber false, DBAccessibleFromOPCUA true, IsOnlyStoredInLoadMemory false, IsRetainMemResEnabled false, IsWriteProtectedInAS false, MemoryReserve 100
   VAR RETAIN
      input : Struct
         "Set Flowrate" : Real;
         "Set time" : DInt;
         "Flowrate adjustment A" : Real;
         "Flowrate adjustment B" : Real;
      END_STRUCT;
   END_VAR
   VAR
      Control : Struct
         "Start metering" : Bool;
         "Stop metering" : Bool;
         "metering running" : Bool;
         "metering completed" : Bool;
      END_STRUCT;
      output : Struct
         "ON_pump A" : Bool;
         "ON_pump B" : Bool;
         ON_mixer : Bool;
         "ON_outlet Valve A" : Bool;
         "Running time" : Int;
         "ON_outlet valve B" : Bool;
         "Volume dispensed" : Real;
         "ON_inlet A" : Bool;
         "ON_inlet B" : Bool;
      END_STRUCT;
   END_VAR
   VAR RETAIN
      "signal type" : Int;
   END_VAR
BEGIN
END_DATA_BLOCK

DATA_BLOCK "Function Dearing with valve"   // DB46
{ S7_Optimized_Access := 'TRUE' }
VERSION : 0.1
// stored: AutoNumber true, DBAccessibleFromOPCUA true, IsOnlyStoredInLoadMemory false, IsRetainMemResEnabled false, IsWriteProtectedInAS false, MemoryReserve 100
   VAR RETAIN
      "Input A" : Struct
         "set time" : Int;
         "set flowrate" : Real;
      END_STRUCT;
      "Input B" : Struct
         "set time" : Int;
         "set flowrate" : Real;
      END_STRUCT;
   END_VAR
   VAR
      "Control A" : Struct
         "start deaaring" : Bool;
         "dearing running" : Bool;
         "stop dearing" : Bool;
         "dearing Completed" : Bool;
      END_STRUCT;
      "Control B" : Struct
         "start deaaring" : Bool;
         "dearing running" : Bool;
         "stop dearing" : Bool;
         "dearing Completed" : Bool;
      END_STRUCT;
      "Output A" : Struct
         "ON pump" : Bool;
         "On outlet valve" : Bool;
         "running time" : Int;
         "ON_inlet A" : Bool;
      END_STRUCT;
      "Output B" : Struct
         "ON pump" : Bool;
         "running time" : Int;
         "On outlet valve" : Bool;
         "ON_inlet B" : Bool;
      END_STRUCT;
   END_VAR
   VAR RETAIN
      "start signal Type" : Int;
   END_VAR
BEGIN
END_DATA_BLOCK

DATA_BLOCK "Function Flush"   // DB47
{ S7_Optimized_Access := 'TRUE' }
VERSION : 0.1
// stored: AutoNumber true, DBAccessibleFromOPCUA true, IsOnlyStoredInLoadMemory false, IsRetainMemResEnabled false, IsWriteProtectedInAS false, MemoryReserve 100
   VAR RETAIN
      Selection : Int;
      "Input A" : Struct
         "set qty" : Real;
         "set flowrate" : Real;
         "Set time" : Int;
         "set time IN MINUTES" : Real;
         "set time in sec" : DInt;
      END_STRUCT;
      "Input B" : Struct
         "set qty" : Real;
         "set flowrate" : Real;
         "Set time" : Int;
         "set time IN MINUTES" : Real;
         "set time in sec" : DInt;
      END_STRUCT;
   END_VAR
   VAR
      "Control A" : Struct
         "Start flushing" : Bool;
         "Stop Flushing" : Bool;
         "flush running" : Bool;
         "flush Completed" : Bool;
      END_STRUCT;
      "Control B" : Struct
         "Start flushing" : Bool;
         "Stop Flushing" : Bool;
         "flush running" : Bool;
         "flush Completed" : Bool;
      END_STRUCT;
      "Output A" : Struct
         "ON pump" : Bool;
         "Running time" : Int;
         "ON  outlet Valve" : Bool;
         "Volume dispensed" : Real;
         "ON_inlet A" : Bool;
      END_STRUCT;
      "Output B" : Struct
         "ON pump" : Bool;
         "Running time" : Int;
         "ON  outlet Valve" : Bool;
         "Volume dispensed" : Real;
         "ON_inlet B" : Bool;
      END_STRUCT;
   END_VAR
   VAR RETAIN
      "Set Qty" : Real;
      Flowrate : Real;
   END_VAR
   VAR
      "AD-HMI" : Struct
         "Set qty" : Real;
         "Set time" : Int;
         "Volume dispensed" : Real;
         "Run time" : Int;
         "Flowrate set" : Real;
      END_STRUCT;
   END_VAR
BEGIN
END_DATA_BLOCK

DATA_BLOCK "Function Metering pgm"   // DB41
{ S7_Optimized_Access := 'TRUE' }
VERSION : 0.1
// stored: AutoNumber true, DBAccessibleFromOPCUA true, IsOnlyStoredInLoadMemory false, IsRetainMemResEnabled false, IsWriteProtectedInAS false, MemoryReserve 100
   VAR RETAIN
      input : Struct
         "Set Flowrate" : Real;
         "Set time" : DInt;
         "Flowrate adjustment A" : Real;
         "Flowrate adjustment B" : Real;
         "set qty" : Real;
      END_STRUCT;
   END_VAR
   VAR
      Control : Struct
         "Start metering" : Bool;
         "Do continuous metering" : Bool;
         "Stop metering" : Bool;
         "metering running" : Bool;
         "metering completed" : Bool;
      END_STRUCT;
      output : Struct
         "ON_pump A" : Bool;
         "ON_pump B" : Bool;
         ON_mixer : Bool;
         "ON_outlet Valve A" : Bool;
         "Running time" : Int;
         "ON_outlet valve B" : Bool;
         "Volume dispensed" : Real;
         "ON_inlet A" : Bool;
         "ON_inlet B" : Bool;
      END_STRUCT;
   END_VAR
BEGIN
END_DATA_BLOCK

DATA_BLOCK "Function Pre run"   // DB42
{ S7_Optimized_Access := 'TRUE' }
VERSION : 0.1
// stored: AutoNumber false, DBAccessibleFromOPCUA true, IsOnlyStoredInLoadMemory false, IsRetainMemResEnabled false, IsWriteProtectedInAS false, MemoryReserve 100
   VAR RETAIN
      input : Struct
         "Set Flowrate" : Real;
         "Set time" : DInt;
         "Flowrate adjustment A" : Real;
         "Flowrate adjustment B" : Real;
         "Pre run Acceleration time" : DInt;
         "Set Qty" : Real;
      END_STRUCT;
   END_VAR
   VAR
      Control : Struct
         "Start metering" : Bool;
         "Stop metering" : Bool;
         "metering running" : Bool;
         "metering completed" : Bool;
      END_STRUCT;
      output : Struct
         "ON_pump A" : Bool;
         "ON_pump B" : Bool;
         ON_mixer : Bool;
         "ON_outlet Valve A" : Bool;
         "Running time" : Int;
         "ON_outlet valve B" : Bool;
         "Volume dispensed" : Real;
         "ON_inlet A" : Bool;
         "ON_inlet B" : Bool;
      END_STRUCT;
   END_VAR
BEGIN
END_DATA_BLOCK

DATA_BLOCK "Function Pressure release"   // DB277
{ S7_Optimized_Access := 'TRUE' }
VERSION : 0.1
// stored: AutoNumber true, DBAccessibleFromOPCUA true, IsOnlyStoredInLoadMemory false, IsRetainMemResEnabled false, IsWriteProtectedInAS false, MemoryReserve 100
   VAR
      "A" : Struct
         Control : Struct
            "Pressure releasing" : Bool;
            "Start release" : Bool;
         END_STRUCT;
         output : Struct
            "ON_outlet Valve A" : Bool;
         END_STRUCT;
      END_STRUCT;
      "B" : Struct
         Control : Struct
            "Start release" : Bool;
            "Pressure releasing" : Bool;
         END_STRUCT;
         output : Struct
            "ON_outlet Valve B" : Bool;
         END_STRUCT;
      END_STRUCT;
      AB : Struct
         Control : Struct
            "Start release" : Bool;
            "Pressure releasing" : Bool;
         END_STRUCT;
         output : Struct
            "ON_outlet Valve B" : Bool;
            "ON_outlet Valve A" : Bool;
         END_STRUCT;
      END_STRUCT;
   END_VAR
BEGIN
END_DATA_BLOCK

DATA_BLOCK "Function Ratio check"   // DB43
{ S7_Optimized_Access := 'TRUE' }
VERSION : 0.1
// stored: AutoNumber false, DBAccessibleFromOPCUA true, IsOnlyStoredInLoadMemory false, IsRetainMemResEnabled false, IsWriteProtectedInAS false, MemoryReserve 100
   VAR RETAIN
      input : Struct
         "Set Flowrate" : Real := 15.0;
         "Set time" : DInt := 0;
         "Flowrate adjustment A" : Real := 0.0;
         "Flowrate adjustment B" : Real := 0.0;
         "set qty" : Real := 1.0;
         Mode : Int := 0;
      END_STRUCT;
   END_VAR
   VAR
      Control : Struct
         "Start metering" : Bool := FALSE;
         "Stop metering" : Bool := FALSE;
         "metering running" : Bool := FALSE;
         "metering completed" : Bool := FALSE;
         "start refill" : Bool := FALSE;
         "quick stop" : Bool := FALSE;
         ProgressBar_Limit : DInt := 4000;
         ProgressBar : DInt := 0;
         AcceptValue : Bool := FALSE;
         ShowPopup : Bool := FALSE;
      END_STRUCT;
      output : Struct
         "ON_pump A" : Bool := FALSE;
         "ON_pump B" : Bool := FALSE;
         ON_mixer : Bool := FALSE;
         "ON_outlet Valve A" : Bool := FALSE;
         "Running time" : Int := 0;
         "ON_outlet valve B" : Bool := FALSE;
         "Volume dispensed" : Real := 0.0;
         "ON_inlet A" : Bool := FALSE;
         "ON_inlet B" : Bool := FALSE;
         "Flowrate running" : Real := 0.0;
         "Remaing qty to dispense" : Real := 0.0;
      END_STRUCT;
   END_VAR
   VAR RETAIN
      PumpCaliberationControls : Struct
         CurrentSet_A : Real := 0.0;
         CurrentSet_B : Real := 0.0;
         CurrentActual_A : Real := 0.0;
         CurrentActual_B : Real := 0.0;
         "CurrentActual_A Gram" : Real := 0.0;
         "CurrentActual_B Gram" : Real := 0.0;
         CurrentSetFlowrate_A : Real := 0.0;
         CurrentSetFlowrate_B : Real := 0.0;
      END_STRUCT;
      PumpCaliberationPara : Struct
         CurrentDeviation_A : Real := 0.0;
         CurrrentDeviation_B : Real := 0.0;
         TotalDeviation_A : Real := 0.0;
         TotalDeviation_B : Real := 0.0;
         "Delete Calibration_A" : Bool := FALSE;
         "Delete Calibration_B" : Bool := FALSE;
      END_STRUCT;
   END_VAR
   VAR
      Parametes : Struct
         AddedMixingRatio : Real := 0.0;
      END_STRUCT;
   END_VAR
BEGIN
END_DATA_BLOCK

DATA_BLOCK "Function Regenaration PGM"   // DB169
{ S7_Optimized_Access := 'TRUE' }
VERSION : 0.1
// stored: AutoNumber false, DBAccessibleFromOPCUA true, IsOnlyStoredInLoadMemory false, IsRetainMemResEnabled false, IsWriteProtectedInAS false, MemoryReserve 100
   VAR RETAIN
      input : Struct
         "Set Flowrate" : Real;
         "Set time" : DInt;
         "Flowrate adjustment A" : Real;
         "Flowrate adjustment B" : Real;
         "set qty" : Real;
      END_STRUCT;
   END_VAR
   VAR
      Control : Struct
         "Start metering" : Bool;
         "Stop metering" : Bool;
         "metering running" : Bool;
         "metering completed" : Bool;
      END_STRUCT;
      output : Struct
         "ON_pump A" : Bool;
         "ON_pump B" : Bool;
         ON_mixer : Bool;
         "ON_outlet Valve A" : Bool;
         "Running time" : Int;
         "ON_outlet valve B" : Bool;
         "Volume dispensed" : Real;
         "ON_inlet A" : Bool;
         "ON_inlet B" : Bool;
      END_STRUCT;
   END_VAR
BEGIN
END_DATA_BLOCK

DATA_BLOCK "Function recirculation"   // DB76
{ S7_Optimized_Access := 'TRUE' }
VERSION : 0.1
// stored: AutoNumber true, DBAccessibleFromOPCUA true, IsOnlyStoredInLoadMemory false, IsRetainMemResEnabled false, IsWriteProtectedInAS false, MemoryReserve 100
   VAR RETAIN
      Selection : Struct
         "A" : Int;
         "B" : Int;
         "A A AB" : Int;
         "A selected" : Bool;
         "B selected" : Bool;
         "A or B selected" : Bool;
      END_STRUCT;
      "recirculation method" : Struct
         "A" : Int;
         "B" : Int;
         "A with Pump" : Bool;
         "B with Pump" : Bool;
         "A or B with Pump" : Bool;
         "A without Pump selected" : Bool;
         "B without Pump selected" : Bool;
      END_STRUCT;
      "time" : Struct
         "active time" : Int;
         "idle time" : Int;
      END_STRUCT;
      Flowrate : Struct
         "A" : Real;
         "B" : Real;
      END_STRUCT;
   END_VAR
   VAR
      "Control A" : Struct
         "start A1" : Bool;
         "start A2" : Bool;
      END_STRUCT;
      "Control B" : Struct
         "start B" : Bool;
      END_STRUCT;
      "Output A1" : Struct
         "ON recirculation valve" : Bool;
         "ON pump" : Bool;
         "On time Done" : Bool;
         Running : Bool;
         Blink : Bool;
      END_STRUCT;
      "Output A2" : Struct
         "ON recirculation valve" : Bool;
         "ON pump" : Bool;
         "On time Done" : Bool;
         Running : Bool;
         Blink : Bool;
      END_STRUCT;
      "Output B1" : Struct
         "ON recirculation valve" : Bool;
         "On time Done" : Bool;
         "ON pump" : Bool;
         Running : Bool;
         Blink : Bool;
      END_STRUCT;
      "time in sec" : Struct
         "active time" : DInt;
         "idle time" : DInt;
      END_STRUCT;
      "A1 time PV" : Struct
         "Active time PV" : Int;
         "Active time PV_ms" : DInt;
         "IDLE time PV_ms" : DInt;
         "IDLE time PV" : Int;
      END_STRUCT;
      "A2 time PV" : Struct
         "Active time PV" : Int;
         "Active time PV_ms" : DInt;
         "IDLE time PV_ms" : DInt;
         "IDLE time PV" : Int;
      END_STRUCT;
      "B1 time PV" : Struct
         "Active time PV" : Int;
         "Active time PV_ms" : DInt;
         "IDLE time PV_ms" : DInt;
         "IDLE time PV" : Int;
      END_STRUCT;
      "AD-HMI A" : Struct
         "set time" : Int;
         "Time PV" : Int;
         "Blink timer" : Bool;
      END_STRUCT;
      "AD-HMI B" : Struct
         "set time" : Int;
         "Time PV" : Int;
         "Blink timer" : Bool;
      END_STRUCT;
   END_VAR
BEGIN
END_DATA_BLOCK

DATA_BLOCK "Function shot Metering"   // DB145
{ S7_Optimized_Access := 'TRUE' }
VERSION : 0.1
// stored: AutoNumber false, DBAccessibleFromOPCUA true, IsOnlyStoredInLoadMemory false, IsRetainMemResEnabled false, IsWriteProtectedInAS false, MemoryReserve 100
   VAR RETAIN
      input : Struct
         "Set Flowrate" : Real;
         "Set time" : DInt;
         "Flowrate adjustment A" : Real;
         "Flowrate adjustment B" : Real;
         "set qty" : Real;
      END_STRUCT;
   END_VAR
   VAR
      Control : Struct
         "Start metering" : Bool;
         "Stop metering" : Bool;
         "metering running" : Bool;
         "metering completed" : Bool;
      END_STRUCT;
      output : Struct
         "ON_pump A" : Bool;
         "ON_pump B" : Bool;
         ON_mixer : Bool;
         "ON_outlet Valve A" : Bool;
         "Running time" : Int;
         "ON_outlet valve B" : Bool;
         "Volume dispensed" : Real;
         "ON_inlet A" : Bool;
         "ON_inlet B" : Bool;
      END_STRUCT;
   END_VAR
BEGIN
END_DATA_BLOCK

DATA_BLOCK "Function_Selection_HMI"   // DB278
{ S7_Optimized_Access := 'TRUE' }
VERSION : 0.1
// stored: AutoNumber true, DBAccessibleFromOPCUA true, IsOnlyStoredInLoadMemory false, IsRetainMemResEnabled false, IsWriteProtectedInAS false, MemoryReserve 100
   VAR
      "Deaering A" : Bool;
      "Deaering B" : Bool;
      "Recirculation A" : Bool;
      "Recirculation B" : Bool;
      Recirculation : Bool;
      "Pressure release A" : Bool;
      "Pressure release B" : Bool;
      "Pressure release" : Bool;
      "Dearing A Without valve" : Bool;
      "Dearing B Without valve" : Bool;
      "Shot metering" : Bool;
      "Continuous metering" : Bool;
      "Metering program" : Bool;
      "Pre run" : Bool;
      "ratio check" : Bool;
      Flush : Bool;
   END_VAR
   VAR RETAIN
      SnuffBack : Bool;
      SnunfBack_flow : Real;
      Snuffback_qty : Real;
   END_VAR
   VAR
      Function_Snuffback_volume_dispensed : Real;
      "Condition Check A" : Bool;
      "Condition Check B" : Bool;
      "Snuffback selected" : Bool;
      "Snuffback start" : Bool;
   END_VAR
BEGIN
END_DATA_BLOCK

DATA_BLOCK "Functions"   // DB40
{ S7_Optimized_Access := 'TRUE' }
VERSION : 0.1
// stored: AutoNumber true, DBAccessibleFromOPCUA true, IsOnlyStoredInLoadMemory false, IsRetainMemResEnabled false, IsWriteProtectedInAS false, MemoryReserve 100
   VAR
      "Dosing function selected" : Bool;
      "Dosing Running" : Bool;
      "Dosing Completed" : Bool;
      "Function running" : Bool;
      "Esc Dosing function" : Bool;
      "Part present R Signal" : Bool;
      "start dosing by partpresent sensor" : Bool;
      "Start Dosing function" : Bool;
      "Start Dosing function site" : Bool;
      "Start dosing function HMI" : Bool;
      "Stop Dosing AB function" : Bool;
      "Stop Dosing B function" : Bool;
      "Stop Dosing A function" : Bool;
      "1k" : Struct
         "deaering A with valve selected" : Bool;
         "deaering B with valve  selected" : Bool;
         "deaering A without valve selected" : Bool;
         "deaering B without valve  selected" : Bool;
         "Flush selected" : Bool;
         "Flush selected during potlife" : Bool;
         "Condition Check A" : Bool;
         "Condition Check B" : Bool;
      END_STRUCT;
      "flush selection" : Struct
         "Flush A selected" : Bool;
         "Flush B selected" : Bool;
         "flush selection in HMI" : Bool;
      END_STRUCT;
      "2k" : Struct
         "metering program selected" : Bool;
         "pre run program selected" : Bool;
         "mixing ratio program selected" : Bool;
         "continous metering program selected" : Bool;
         "shot metering program selected" : Bool;
         "regeration program selected" : Bool;
      END_STRUCT;
      "Block all 1k metering" : Bool;
      "Block all 2k metering" : Bool;
      "Deselect all function" : Bool;
      "recirculation Selected" : Bool;
      "Pressure release selected" : Bool;
      "recirculation A selected" : Bool;
      "recirculation B selected" : Bool;
      "Pressure release A selected" : Bool;
      "Pressure release B selected" : Bool;
      "Stop Dosing function" : Bool;
      "stop dosing function site" : Bool;
      Functions : Int;
   END_VAR
   VAR RETAIN
      Auto : Bool;
   END_VAR
BEGIN
END_DATA_BLOCK

DATA_BLOCK "HMI"   // DB1
{ S7_Optimized_Access := 'TRUE' }
VERSION : 0.1
// stored: AutoNumber true, DBAccessibleFromOPCUA true, IsOnlyStoredInLoadMemory false, IsRetainMemResEnabled false, IsWriteProtectedInAS false, MemoryReserve 100
   VAR
      "screen no to change" : Int;
      unit : Struct
         cm3 : Int;
         cm3_min : Int;
         ml : Int;
         ml_min : Int;
         "degree celsius" : Int;
         precentage : Int;
         seonds : Int;
         minutes : Int;
         hours : Int;
         bar : Int;
         mbar : Int;
         milliseconds : Int;
         RPM : Int;
         imp : Int;
         "cm3/r" : Int;
         set : Int;
         "real" : Int;
         "type" : Int;
         day : Int;
         "cm3/imp" : Int;
         "imp/rev" : Int;
         "m" : Int;
      END_STRUCT;
      "A" : Int;
      "B" : Int;
      "Screen no by function" : Int;
      "Current screen No" : Int;
      "Function ONS" : Struct
         "Dearing A" : Bool;
         "function deselected" : Bool;
         "Dearing B" : Bool;
         "Dearing A coil" : Bool;
         "dearing B Coil" : Bool;
         Flush : Bool;
         "pre run" : Bool;
         "Ratio Check" : Bool;
         "Shot metering Program" : Bool;
         "Continous metering prgram" : Bool;
         "metering program" : Bool;
         "recirculation A" : Bool;
         "recirculation B" : Bool;
         Recirculation : Bool;
         "pressure release A" : Bool;
         "pressure release B" : Bool;
         "Pressure release AB" : Bool;
         regeneration : Bool;
         "flush potlife" : Bool;
         "checkConditionA Coil" : Bool;
         "checkConditionB Coil" : Bool;
         checkConditionA : Bool;
         checkConditionB : Bool;
      END_STRUCT;
      "HMI User" : WString;
      AdminLogged : Bool;
      userlogged : Bool;
      "HMI user To hmi" : WString;
   END_VAR
   VAR RETAIN
      supplySelection : Int;
   END_VAR
BEGIN
END_DATA_BLOCK

DATA_BLOCK "IOT_DATA"   // DB1001
{ S7_Optimized_Access := 'FALSE' }
VERSION : 0.1
// stored: AutoNumber false, DBAccessibleFromOPCUA true, IsOnlyStoredInLoadMemory false, IsWriteProtectedInAS false
   VAR
      "pump A Inlet" { ExternalAccessible := 'False'; ExternalVisible := 'False'; ExternalWritable := 'False'} : Real;
      "pump B Inlet" { ExternalAccessible := 'False'; ExternalVisible := 'False'; ExternalWritable := 'False'} : Real;
      "pump A Outlet" { ExternalAccessible := 'False'; ExternalVisible := 'False'; ExternalWritable := 'False'} : Real;
      "pump B Outlet" { ExternalAccessible := 'False'; ExternalVisible := 'False'; ExternalWritable := 'False'} : Real;
   END_VAR
BEGIN
END_DATA_BLOCK

DATA_BLOCK "Machine infromation"   // DB80
{ S7_Optimized_Access := 'TRUE' }
VERSION : 0.1
// stored: AutoNumber true, DBAccessibleFromOPCUA true, IsOnlyStoredInLoadMemory false, IsRetainMemResEnabled false, IsWriteProtectedInAS false, MemoryReserve 100
   VAR RETAIN
      "Software No" : String := 'P-761.V0 20220930';
   END_VAR
BEGIN
END_DATA_BLOCK

DATA_BLOCK "Material Data current pgm"   // DB330
{ S7_Optimized_Access := 'TRUE' }
VERSION : 0.1
// stored: AutoNumber true, DBAccessibleFromOPCUA true, IsOnlyStoredInLoadMemory false, IsRetainMemResEnabled false, IsWriteProtectedInAS false, MemoryReserve 100
   VAR RETAIN
      Density : Struct
         "A" : Real;
         "B" : Real;
      END_STRUCT;
      Viscosity : Struct
         "A" : Real;
         "B" : Real;
      END_STRUCT;
      "Name" : Struct
         "A" : String[20];
         "B" : String[20];
      END_STRUCT;
      "name A+B" : String[40];
      "Mixed Density" : Real;
      BatchA : String[20];
      BatchB : String[20];
      "+symbol" : String := '+';
   END_VAR
BEGIN
END_DATA_BLOCK

DATA_BLOCK "Metering Program Parameters"   // DB45
{ S7_Optimized_Access := 'FALSE' }
VERSION : 0.1
// stored: AutoNumber true, DBAccessibleFromOPCUA true, IsOnlyStoredInLoadMemory false, IsWriteProtectedInAS false
   VAR RETAIN
      "program No site" : Int;
      "Program No screen" : Int;
      "Receipe Program No" : DInt;
      "Receipe Set Flowrate" : Real;
      "Receipe Set qty" : Real;
      "Receipe Description" : String[12];
      "Receipe Flowrate Adjustment A" : Real;
      "Receipe Flowrate Adjustment B" : Real;
      "Current Program" : Struct
         "Set Flowrate" : Real;
         "Set qty" : Real;
         Description : String[12];
         "Flowrate Adjustment A" : Real;
         "Flowrate Adjustment B" : Real;
         "Set Flowrate snuffback" : Real;
         "Set qty snuffback" : Real;
         "Set delay snuffback" : Time;
      END_STRUCT;
      "Current program No" : DInt;
      "Min Mixed Flowrate Ml" : Real;
      "Max Mixed Flowrate Ml" : Real;
      "Max A Flowrate Ml" : Real;
      "Max B Flowrate Ml" : Real;
      "Receipe Set Flowrate snuffback" : Real;
      "Receipe Set Qty snuffback" : Real;
      "Receipe Set delay snuffback" : Time;
   END_VAR
BEGIN
END_DATA_BLOCK

DATA_BLOCK "Metering control"   // DB116
{ S7_Optimized_Access := 'TRUE' }
VERSION : 0.1
// stored: AutoNumber true, DBAccessibleFromOPCUA true, IsOnlyStoredInLoadMemory false, IsRetainMemResEnabled false, IsWriteProtectedInAS false, MemoryReserve 100
   VAR RETAIN
      "outlet valve" : Struct
         selection : Int;
         "common selected" : Bool;
         individual : Bool;
      END_STRUCT;
      Reneration : Struct
         selection : Int := 1;
         selected : Bool;
      END_STRUCT;
      Flush : Struct
         selection : Int;
         selected : Bool;
      END_STRUCT;
      compression : Struct
         selection : Int;
         selected : Bool;
      END_STRUCT;
      Refilling : Struct
         "selection A" : Int;
         "selection B" : Int;
      END_STRUCT;
      "system Preparation" : Struct
         "A selection" : Int := 1;
         "B selection" : Int := 1;
      END_STRUCT;
      "Ready to meter" : Struct
         "pressure less selection A" : Int := 1;
         "Pressure less selection  B" : Int := 1;
         "Heater interlock" : Bool;
      END_STRUCT;
   END_VAR
BEGIN
END_DATA_BLOCK

DATA_BLOCK "Metering"   // DB5
{ S7_Optimized_Access := 'TRUE' }
VERSION : 0.1
// stored: AutoNumber true, DBAccessibleFromOPCUA true, IsOnlyStoredInLoadMemory false, IsRetainMemResEnabled false, IsWriteProtectedInAS false, MemoryReserve 100
   VAR
      Metering_start : Bool;
      Metering_stop : Bool;
      Metering_completed : Bool;
      Metering_running : Bool;
   END_VAR
   VAR RETAIN
      input : Struct
         "Set Flowrate" : Real;
         "Set time" : DInt;
         "Flowrate adjustment A" : Real;
         "Flowrate adjustment B" : Real;
      END_STRUCT;
   END_VAR
   VAR
      Control : Struct
         "Start metering" : Bool;
         "Stop metering" : Bool;
         "metering running" : Bool;
         "metering completed" : Bool;
      END_STRUCT;
      output : Struct
         "ON_pump A" : Bool;
         "ON_pump B" : Bool;
         ON_mixer : Bool;
         "ON_outlet Valve A" : Bool;
         "Running time" : Int;
         "ON_outlet valve B" : Bool;
         "Volume dispensed" : Real;
         "ON_inlet A" : Bool;
         "ON_inlet B" : Bool;
      END_STRUCT;
   END_VAR
BEGIN
END_DATA_BLOCK

DATA_BLOCK "Mixing ratio"   // DB70
{ S7_Optimized_Access := 'TRUE' }
VERSION : 0.1
// stored: AutoNumber true, DBAccessibleFromOPCUA true, IsOnlyStoredInLoadMemory false, IsRetainMemResEnabled false, IsWriteProtectedInAS false, MemoryReserve 100
   VAR RETAIN
      "Mixing ratio according to density" : Real;
      "Mixing ratio set" : Real;
      "Mixing ratio tolerence for error" : Real;
      "Mixing ratio tolerence for warning" : Real;
   END_VAR
   VAR
      "Check MR" : Bool;
      "check mr0" : Bool;
      "Check MR ONS" : Bool;
      "Ratio check done" : Bool;
   END_VAR
   VAR RETAIN
      "MR check delay start time" : Int;
   END_VAR
   VAR
      "MR PV" : Real;
      "MR deviation" : Real;
      "Mixing ratio high Error" : Bool;
      "mixing ratio high Warning" : Bool;
      "Mixing ratio Low  Error" : Bool;
      "mixing ratio Low Warning" : Bool;
      "Mixing ratio Okay" : Bool;
      "Mixing ratio check done" : Bool;
      "mixing ratio check delay in Sec" : DInt;
      "ratio Min" : Real;
      "ratio max" : Real;
      "Mixing ratio Okay On recirculation" : Bool;
      "Mixing ratio error during recirculation" : Bool;
   END_VAR
BEGIN
END_DATA_BLOCK

DATA_BLOCK "PID_correction"   // DB350
{ S7_Optimized_Access := 'TRUE' }
VERSION : 0.1
// stored: AutoNumber false, DBAccessibleFromOPCUA true, IsOnlyStoredInLoadMemory false, IsRetainMemResEnabled false, IsWriteProtectedInAS false, MemoryReserve 100
   VAR
      "Flowrate withadjustment" : Struct
         "A" : Real;
         "B" : Real;
      END_STRUCT;
      "Flowrate with adjustment_ml" : Struct
         "A" : Real;
         "B" : Real;
      END_STRUCT;
      "Manual Value" : Struct
         "A" : Real;
         "B" : Real;
      END_STRUCT;
      "Flowrate%" : Struct
         "A" : Real;
         "B" : Real;
      END_STRUCT;
      "Start manual Mode" : Struct
         "A" : Bool;
         "B" : Bool;
      END_STRUCT;
      "Start Auto Mode" : Struct
         "A" : Bool;
         "B" : Bool;
      END_STRUCT;
   END_VAR
BEGIN
END_DATA_BLOCK

DATA_BLOCK "Pid Control A"   // DB311
{ S7_Optimized_Access := 'TRUE' }
VERSION : 0.1
// stored: AutoNumber false, DBAccessibleFromOPCUA true, IsOnlyStoredInLoadMemory false, IsRetainMemResEnabled false, IsWriteProtectedInAS false, MemoryReserve 100
   VAR
      input : Struct
         setflowrate : Real;
         "Flowrate input" : Real;
         "current flowrate" : Real;
         "Ramp up rate" : Real;
         start : Bool;
         "delay time On" : Bool;
         "setflowrate Low" : Real;
         "setflowrate high" : Real;
         "output low" : Real;
         "output high" : Real;
         "input low" : Real;
         "input high" : Real;
      END_STRUCT;
   END_VAR
   VAR RETAIN
      Control : Struct
         P : Real;
         i : Real;
         d : Real;
         "rampup time" : Real;
         "Activate manual mode" : Bool;
         "Start Delay time" : DInt;
      END_STRUCT;
   END_VAR
   VAR
      Output : Struct
         "output percentage" : Real;
      END_STRUCT;
      Misc : Struct
         error : Bool;
         "error bits" : Int;
         states : Int;
      END_STRUCT;
   END_VAR
   VAR RETAIN
      Enable : Int;
   END_VAR
BEGIN
END_DATA_BLOCK

DATA_BLOCK "Pid Control B"   // DB312
{ S7_Optimized_Access := 'TRUE' }
VERSION : 0.1
// stored: AutoNumber false, DBAccessibleFromOPCUA true, IsOnlyStoredInLoadMemory false, IsRetainMemResEnabled false, IsWriteProtectedInAS false, MemoryReserve 100
   VAR
      input : Struct
         setflowrate : Real;
         "Flowrate input" : Real;
         "current flowrate" : Real;
         "Ramp up rate" : Real;
         start : Bool;
         "delay time On" : Bool;
         "setflowrate Low" : Real;
         "setflowrate high" : Real;
         "output low" : Real;
         "output high" : Real;
         "input low" : Real;
         "input high" : Real;
      END_STRUCT;
   END_VAR
   VAR RETAIN
      Control : Struct
         P : Real;
         i : Real;
         d : Real;
         "rampup time" : Real;
         "start Delay time" : DInt;
         "Activate manual mode" : Bool;
      END_STRUCT;
   END_VAR
   VAR
      Output : Struct
         "output percentage" : Real;
      END_STRUCT;
      Misc : Struct
         error : Bool;
         "error bits" : Int;
         states : Int;
      END_STRUCT;
   END_VAR
   VAR RETAIN
      Enable : Int;
   END_VAR
BEGIN
END_DATA_BLOCK

DATA_BLOCK "Pop-up Db"   // DB341
{ S7_Optimized_Access := 'TRUE' }
VERSION : 0.1
// stored: AutoNumber true, DBAccessibleFromOPCUA true, IsOnlyStoredInLoadMemory false, IsRetainMemResEnabled false, IsWriteProtectedInAS false, MemoryReserve 100
   VAR
      "Additional metering Popup-enable" : Bool;
      "Close Button" : Bool;
      "General Visibility" : Bool;
      "Dearing A Visibility" : Bool;
      "Dearing B Visibility" : Bool;
      "Dearing C Visibility" : Bool;
      "Condition check visibility" : Bool;
   END_VAR
   VAR RETAIN
      parameter_scrno_condchecken : String[2];
   END_VAR
BEGIN
END_DATA_BLOCK

DATA_BLOCK "Potlife"   // DB73
{ S7_Optimized_Access := 'TRUE' }
VERSION : 0.1
// stored: AutoNumber true, DBAccessibleFromOPCUA true, IsOnlyStoredInLoadMemory false, IsRetainMemResEnabled false, IsWriteProtectedInAS false, MemoryReserve 100
   VAR
      "run time" : Struct
         Hours : Int := 0;
         minutes : Int := 0;
         seconds : Int := 0;
      END_STRUCT;
   END_VAR
   VAR RETAIN
      "set time format" : Int := 0;
      "enable potlife" : Int := 0;
   END_VAR
   VAR
      "potlife life enabled" : Bool := FALSE;
   END_VAR
   VAR RETAIN
      "set time" : Int := 30;
   END_VAR
   VAR
      "Potlife time in seconds" : Bool := FALSE;
      "potlife time in minutes" : Bool := TRUE;
   END_VAR
   VAR RETAIN
      "Mixing Volume to dispense" : Real := 3.0;
      Flowrate : Real := 3.0;
      "Control time" : Int := 60;
   END_VAR
   VAR
      "Control time in sec" : DInt := -5536;
   END_VAR
   VAR RETAIN
      "Maximum number of cycle" : Int := 5;
   END_VAR
   VAR
      "potlifetime format" : Int := 0;
      "set time input" : Struct
         seconds : DInt := 30000;
         minutes : DInt := 1800000;
      END_STRUCT;
      contol : Struct
         "trigger potlife" : Bool := TRUE;
         "Potlife elapsed Start Regeneration" : Bool := TRUE;
         "start potlife timer" : Bool := TRUE;
         "Seconds timer Done" : Bool := FALSE;
         "minutes timer Done" : Bool := TRUE;
         "60sec pulse done" : Bool := FALSE;
         "reset counter" : Bool := TRUE;
         "Potlife elapsed machine not in regeneration" : Bool := TRUE;
         "start reneration program" : Bool := FALSE;
         "Start Sequence" : Bool := FALSE;
      END_STRUCT;
      "Time PV" : Struct
         "Sectimer PV" : DInt := 0;
         minutestimerPV : DInt := 1800000;
         "secPulse PV" : Int := 0;
      END_STRUCT;
      "Time PV unscalled" : Struct
         "Sectimer PV" : Int := 0;
         minutestimerPV : Int := 30;
         "secPulse PV" : Int := 0;
      END_STRUCT;
      "Time PV Down Counts" : Struct
         "Sectimer PV" : DInt := 0;
         minutestimerPV : DInt := 0;
         "secPulse PV" : Int := 0;
      END_STRUCT;
      "Flush Control" : Struct
         "maximum cycle reached" : Bool := FALSE;
         "Flush pgm selected" : Bool := FALSE;
         "start Flush" : Bool := FALSE;
      END_STRUCT;
      "Control time in sec_1" : DInt;
   END_VAR
BEGIN
END_DATA_BLOCK

DATA_BLOCK "Pump & Flowrate"   // DB48
{ S7_Optimized_Access := 'TRUE' }
VERSION : 0.1
// stored: AutoNumber true, DBAccessibleFromOPCUA true, IsOnlyStoredInLoadMemory false, IsRetainMemResEnabled false, IsWriteProtectedInAS false, MemoryReserve 100
   VAR RETAIN
      "Pump A" : Struct
         size : Real := 0.0590186;
         "Pump Speed" : Int := 200;
         "speed sensor impulse" : Int := 0;
         "size in ml" : Real := 0.0590186;
         "serial number" : String[20] := '';
      END_STRUCT;
      "Pump B" : Struct
         size : Real := 0.0546615;
         "size in ml" : Real := 0.0546615;
         "Pump Speed" : Int := 200;
         "speed sensor impulse" : Int := 0;
         "serial number" : String[20] := '';
      END_STRUCT;
   END_VAR
   VAR
      capacity : Struct
         "Pump A" : Real := 11.80372;
         "pump B in ml" : Real := 10.9323;
         "pump A in ml" : Real := 11.80372;
         "pump B" : Real := 10.9323;
      END_STRUCT;
      "Flowrate Input" : Struct
         "Pump A" : Real := 5.0;
         "Pump A in ml" : Real := 5.0;
         "pump B in ml" : Real := 2.0;
         "Pump B" : Real := 2.0;
      END_STRUCT;
      "mixed flowrate Input" : Real := 6.0;
      "Qty input" : Real := 0.5;
      "Calculated flowrate A with adjustment" : Real := 4.0;
      "Calculated Flowrate B  with adjustment" : Real := 2.0;
      "Calculated flowrate A without adjustment" : Real := 4.0;
      "Calculated Flowrate B without adjustment" : Real := 2.0;
      "Flowrate Adjustment A" : Real := 0.0;
      "Flowrate Adjustment B" : Real := 0.0;
      "Metering time calculated" : DInt := 5000;
      "Mixed Flowrate maximum" : Real := 0.0;
      "metering time in seconds" : Int := 5;
      "fowrate A Adjustment Configuration" : Real := 0.0;
      "fowrate B Adjustment Configuration" : Real := 0.0;
      "Maximum Mixed Flowrate" : Real := 17.70558;
      "Minimum Mixed Flowrate" : Real := 0.1062335;
      "Pump A minimum Flowrate" : Real := 1.180372;
      "Pump B minimum Flowrate" : Real := 1.09323;
      "Flush Maximum Flowrate" : Real := 10.9323;
      "Flush minimum Flowrate" : Real := 1.09323;
      startSnuff_Back_PumpA : Bool := TRUE;
      startSnuff_Back_PumpB : Bool := TRUE;
      SnuffBack_SpeedA : Bool := FALSE;
   END_VAR
   VAR RETAIN
      referenceRamp_PumpA : Real := 6000.0;
      referenceRamp_PumpB : Real := 6000.0;
      PumpsizeA_original : Real := 0.05;
      PumpsizeB_original : Real := 0.05;
   END_VAR
   VAR
      pumpA_edited : Bool := FALSE;
      pumpB_edited : Bool := FALSE;
      record_size : Bool := FALSE;
   END_VAR
BEGIN
END_DATA_BLOCK

DATA_BLOCK "Pump Manage"   // DB307
{ S7_Optimized_Access := 'TRUE' }
VERSION : 0.1
// stored: AutoNumber true, DBAccessibleFromOPCUA true, IsOnlyStoredInLoadMemory false, IsRetainMemResEnabled false, IsWriteProtectedInAS false, MemoryReserve 100
   VAR RETAIN
      "Pump A-Run Time Hours<50%" : UDInt;
      "Pump A-Run Time Minuts<50%" : UDInt;
      "Pump A-Run Time Seconds<50%" : UDInt;
      "Pump B-Run Time Hours<50%" : UDInt;
      "Pump B-Run Time Minuts<50%" : UDInt;
      "Pump B-Run Time Seconds<50%" : UDInt;
      "Pump A-Run Time Hours>50%" : UDInt;
      "Pump A-Run Time Minuts>50%" : UDInt;
      "Pump A-Run Time Seconds>50%" : UDInt;
      "Pump B-Run Time Hours>50%" : UDInt;
      "Pump B-Run Time Minuts>50%" : UDInt;
      "Pump B-Run Time Seconds>50%" : UDInt;
   END_VAR
   VAR
      "Pump A Min Reset<50" : Bool;
      "Pump A Hrs Reset1<50" : Bool;
      "comm Pump A Hrs Reset<50" : Bool;
      "Pump A Hrs Reset<50" : Bool;
      "Pump A Sec Reset<50" : Bool;
      "Pump A Min Reset>50" : Bool;
      "Pump A Hrs Reset>50" : Bool;
      "Pump A Hrs Reset1>50" : Bool;
      "comm Pump A Hrs Reset>50" : Bool;
      "Pump A Sec Reset>50" : Bool;
      "Pump B Min Reset<50" : Bool;
      "Pump B Hrs Reset<50" : Bool;
      "Pump B Hrs Reset1<50" : Bool;
      "comm Pump B Hrs Reset<50" : Bool;
      "Pump B Sec Reset<50" : Bool;
      "Pump B Min Reset>50" : Bool;
      "Pump B Hrs Reset>50" : Bool;
      "Pump B Hrs Reset1>50" : Bool;
      "comm Pump B Hrs Reset>50" : Bool;
      "Pump B Sec Reset>50" : Bool;
      "Reset A pump Hours and Minutes" : Bool;
      "Reset B pump Hours and Minutes" : Bool;
   END_VAR
   VAR RETAIN
      "Pump A Total Run Hours" : UDInt;
      "Pump B Total Run Hours" : UDInt;
      "Pump A Total Run Minutes" : UDInt;
      "Pump B Total Run Minutes" : UDInt;
   END_VAR
   VAR
      "Pump SEc Reset" : Struct
         "comm Pump A Sec Reset<50" : Bool;
         "comm Pump A Sec Reset>50" : Bool;
         "comm Pump B Sec Reset<50" : Bool;
         "comm Pump B Sec Reset>50" : Bool;
      END_STRUCT;
   END_VAR
BEGIN
END_DATA_BLOCK

DATA_BLOCK "RPM"   // DB77
{ S7_Optimized_Access := 'TRUE' }
VERSION : 0.1
// stored: AutoNumber true, DBAccessibleFromOPCUA true, IsOnlyStoredInLoadMemory false, IsRetainMemResEnabled false, IsWriteProtectedInAS false, MemoryReserve 100
   VAR
      "A" : Real;
      "B" : Real;
   END_VAR
   VAR RETAIN
      "speed sensor selection A" : Int;
      "speed sensor selection B" : Int;
   END_VAR
   VAR
      "a selected" : Bool;
      "b selected" : Bool;
      "ab selected" : Bool;
      "No signal RPM sensor A" : Bool;
      "No signal RPM sensor B" : Bool;
      "A frequency" : Real;
      "B frequency" : Real;
   END_VAR
BEGIN
END_DATA_BLOCK

DATA_BLOCK "Re-filling Sequence DB"   // DB103
{ S7_Optimized_Access := 'TRUE' }
VERSION : 0.1
// stored: AutoNumber true, DBAccessibleFromOPCUA true, IsOnlyStoredInLoadMemory false, IsRetainMemResEnabled false, IsWriteProtectedInAS false, MemoryReserve 100
   VAR
      "Refilling Enable" : Bool;
      "Refilling manual Comp A" : Bool;
      "Refilling manual Comp B" : Bool;
      "Refiling ValveA ON" : Bool;
      "Refiling ValveA ON Manual" : Bool;
      "Refilling Manual Componet A" : Bool;
      "Refilling Manual Componet B" : Bool;
      "Refiling ValveB ON" : Bool;
      "Refiling ValveB ON Manual" : Bool;
      "AODD Pump Component A ON" : Bool;
      "AODD Pump Component A ON- Manual" : Bool;
      "AODD Pump Component B ON" : Bool;
      "AODD Pump Component B ON- Manual" : Bool;
   END_VAR
   VAR RETAIN
      "AODD  componet A  ON delay" : Time;
      "AODD  componet B  ON delay" : Time;
   END_VAR
   VAR
      "Compare Re-fillingFilling sequence A" : Struct
         "Start Compare" : Bool;
         "Re-filling % in 30 Sec" : Real;
         "Excpected Level" : Real;
         "Refilling Error" : Bool;
      END_STRUCT;
      "Compare Filling sequence b" : Struct
         "Start Compare" : Bool;
         "Re-filling % in 30 Sec" : Real;
         "Excpected Level" : Real;
         "Refilling Error" : Bool;
      END_STRUCT;
   END_VAR
   VAR RETAIN
      "A valve off pump off delay" : DInt;
      "B valve off pump off delay" : DInt;
   END_VAR
   VAR
      temp1 : Bool;
      temp2 : Bool;
   END_VAR
BEGIN
END_DATA_BLOCK

DATA_BLOCK "Refilling"   // DB136
{ S7_Optimized_Access := 'TRUE' }
VERSION : 0.1
// stored: AutoNumber true, DBAccessibleFromOPCUA true, IsOnlyStoredInLoadMemory false, IsRetainMemResEnabled false, IsWriteProtectedInAS false, MemoryReserve 100
   VAR
      Running : Struct
         A1 : Bool;
         A2 : Bool;
         B1 : Bool;
      END_STRUCT;
      "Control A1" : Struct
         "Start Refilling" : Bool;
         "refilling failed" : Bool;
      END_STRUCT;
      "Control A2" : Struct
         "Start Refilling" : Bool;
         "refilling failed" : Bool;
      END_STRUCT;
      "Control B1" : Struct
         "Start Refilling" : Bool;
         "refilling failed" : Bool;
      END_STRUCT;
      "Output A1" : Struct
         "Run vacuum PUMP" : Bool;
         "Open Vaccum Valve" : Bool;
         "Open refilling Valve" : Bool;
         "Pump minimum run time okay" : Bool;
      END_STRUCT;
      "Output A2" : Struct
         "Run vacuum PUMP" : Bool;
         "Open Vaccum Valve" : Bool;
         "Open refilling Valve" : Bool;
         "Pump minimum run time okay" : Bool;
      END_STRUCT;
      "Output B1" : Struct
         "Run vacuum PUMP" : Bool;
         "Open Vaccum Valve" : Bool;
         "Open refilling Valve" : Bool;
         "Pump minimum run time okay" : Bool;
      END_STRUCT;
      "filling level A1" : Struct
         "Filling level reached" : Bool;
         "Filling failed" : Bool;
         "Previous value" : Real;
         "current value" : Real;
         "start Compare" : Bool;
         "stop compare" : Bool;
      END_STRUCT;
      "filling level A2" : Struct
         "Filling level reached" : Bool;
         "Filling failed" : Bool;
         "Previous value" : Real;
         "current value" : Real;
         "start Compare" : Bool;
         "stop compare" : Bool;
      END_STRUCT;
      "filling level B1" : Struct
         "Filling level reached" : Bool;
         "Filling failed" : Bool;
         "Previous value" : Real;
         "current value" : Real;
         "start Compare" : Bool;
         "stop compare" : Bool;
      END_STRUCT;
   END_VAR
   VAR RETAIN
      "level increase in 30s" : Struct
         "A" : Real;
         "B" : Real;
      END_STRUCT;
      PressureExaustTime : DInt;
   END_VAR
   VAR
      PressureReleaseA : Bool;
      PressureReleaseB : Bool;
      "Start Auto Refill A" : Bool;
      "Start Auto Refill B" : Bool;
   END_VAR
   VAR RETAIN
      PressureExaustTimeS : DInt;
   END_VAR
   VAR
      Temp1 : Bool;
      Temp2 : Bool;
   END_VAR
BEGIN
END_DATA_BLOCK

DATA_BLOCK "Servo Control"   // DB336
{ S7_Optimized_Access := 'TRUE' }
VERSION : 0.1
// stored: AutoNumber false, DBAccessibleFromOPCUA true, IsOnlyStoredInLoadMemory false, IsRetainMemResEnabled false, IsWriteProtectedInAS false, MemoryReserve 100
   VAR
      "A" : Struct
         "Power On" : Bool;
         Reset : Bool;
         Restart : Bool;
         "Speed input" : Real;
         Velocity : Real;
         "Power Error" : Bool;
         "drive error" : Bool;
         "Communication Error" : Bool;
         "Actual Velocity" : Real;
         RPM : Real;
      END_STRUCT;
      "B" : Struct
         "Power On" : Bool;
         Reset : Bool;
         Restart : Bool;
         "Speed input" : Real;
         Velocity : Real;
         "Power Error" : Bool;
         "drive error" : Bool;
         "Communication Error" : Bool;
         "Actual Velocity" : Real;
         RPM : Real;
      END_STRUCT;
      Mixer : Struct
         "Power On" : Bool;
         Reset : Bool;
         Restart : Bool;
         "Speed input" : Real;
         Velocity : Real;
         "Power Error" : Bool;
         "drive error" : Bool;
         "Communication Error" : Bool;
         "Actual Velocity" : Real;
         RPM : Real;
      END_STRUCT;
   END_VAR
BEGIN
END_DATA_BLOCK

DATA_BLOCK "Temp"   // DB167
{ S7_Optimized_Access := 'TRUE' }
VERSION : 0.1
// stored: AutoNumber true, DBAccessibleFromOPCUA true, IsOnlyStoredInLoadMemory false, IsRetainMemResEnabled false, IsWriteProtectedInAS false, MemoryReserve 100
   VAR
      bit1 : Bool;
      bit2 : Bool;
      bit3 : Bool;
      bit4 : Bool;
      bit5 : Bool;
      bit6 : Bool;
      bit7 : Bool;
      bit8 : Bool;
      bit9 : Bool;
      bit10 : Bool;
      bit11 : Bool;
      bit12 : Bool;
      bit13 : Bool;
      bit14 : Bool;
      bit15 : Bool;
      bit16 : Bool;
      bit17 : Bool;
      bit18 : Bool;
      bit19 : Bool;
      bit20 : Bool;
      bit21 : Bool;
      bit22 : Bool;
      bit23 : Bool;
      bit24 : Bool;
      bit25 : Bool;
      bit26 : Bool;
      bit27 : Bool;
      temp : Int;
      temp_1 : Int;
      temp_2 : Int;
      temp_3 : Array[0..30] of Bool;
   END_VAR
   VAR RETAIN
      Snuffback_ONdelay_A : Time := T#5MS;
      Snuffback_OFFdelay_A : Time := T#5MS;
      Snuffback_Ondelay_B : Time := T#1S;
      Snuffback_OFFdelay_B : Time := T#1S;
   END_VAR
   VAR
      Snuffback_vol_dispensedA { ExternalAccessible := 'False'; ExternalVisible := 'False'; ExternalWritable := 'False'} : Real;
      Snuffback_vol_dispensedB { ExternalAccessible := 'False'; ExternalVisible := 'False'; ExternalWritable := 'False'} : Real;
      Metering_time_inSec { ExternalAccessible := 'False'; ExternalVisible := 'False'; ExternalWritable := 'False'} : Time;
   END_VAR
   VAR RETAIN
      Language_selection : Int;
   END_VAR
   VAR
      temp_4 : Array[0..10] of Bool;
      ratiocheck_temp : Array[0..10] of Bool;
   END_VAR
BEGIN
END_DATA_BLOCK

DATA_BLOCK "VC_pulseHMI"   // DB344
{ S7_Optimized_Access := 'TRUE' }
VERSION : 0.1
// stored: AutoNumber true, DBAccessibleFromOPCUA true, IsOnlyStoredInLoadMemory false, IsRetainMemResEnabled false, IsWriteProtectedInAS false, MemoryReserve 100
   VAR
      "current Pulse VC1" : DInt;
      "current Pulse VC2" : DInt;
      "Previous Pulse VC1" : DInt;
      "Previous Pulse VC2" : DInt;
      "reset VC1" : Bool;
      "reset VC2" : Bool;
   END_VAR
BEGIN
END_DATA_BLOCK

DATA_BLOCK "Volume counter"   // DB206
{ S7_Optimized_Access := 'TRUE' }
VERSION : 0.1
// stored: AutoNumber true, DBAccessibleFromOPCUA true, IsOnlyStoredInLoadMemory false, IsRetainMemResEnabled false, IsWriteProtectedInAS false, MemoryReserve 100
   VAR RETAIN
      "A" : Struct
         Impulse : Real := 0.0;
         "Impulse in HMI" : Real := 0.00625;
         "Maximum Down time" : Int;
         "Maximum Down time in sec" : DInt;
         "serial number" : String;
         "Leakage Pulses" : Int;
         "Leakage Control time" : Int;
         "Leakage control time in Sec" : DInt;
      END_STRUCT;
      "B" : Struct
         Impulse : Real;
         "Impulse in HMI" : Real := 0.00625;
         "Maximum Down time" : Int;
         "Maximum Down time in sec" : DInt;
         "serial number" : String;
         "Leakage Pulses" : Int;
         "Leakage Control time" : Int;
         "Leakage control time in Sec" : DInt;
      END_STRUCT;
   END_VAR
   VAR
      "Control A" : Struct
         "Create CV during Process" : Bool;
         "New CV during Process" : DInt;
         "Current Pulses during process" : DInt;
         "Create New CV For ratio check" : Bool;
         "New CV  For ratio check" : DInt;
         "Current Pulses  For ratio check" : DInt;
      END_STRUCT;
      "Control B" : Struct
         "Create CV during Process" : Bool;
         "New CV during Process" : DInt;
         "Current Pulses during process" : DInt;
         "Create New CV For ratio check" : Bool;
         "New CV For ratio check" : DInt;
         "Current Pulses For ratio check" : DInt;
      END_STRUCT;
      "Volume A" : Struct
         "volume For Ratio check" : Real;
         "volume For Qty Display" : Real;
      END_STRUCT;
      "Volume B" : Struct
         "volume For Ratio check" : Real;
         "volume For Qty Display" : Real;
      END_STRUCT;
      Volume : Struct
         "For Process" : Real;
         "For Ratio Check" : Real;
      END_STRUCT;
      "Process running start volume measurement" : Bool;
      "Process running start volume measurement ONS" : Bool;
   END_VAR
   VAR RETAIN
      Selection : Struct
         "A" : Int := 0;
         "B" : Int := 0;
      END_STRUCT;
      Enabled : Struct
         "A" : Bool;
         "B" : Bool;
         AB : Bool;
      END_STRUCT;
   END_VAR
   VAR
      "No signal" : Struct
         "A" : Bool;
         "B" : Bool;
      END_STRUCT;
      "Leakage Control A" : Struct
         "Start Test" : Bool;
         "Start Test ONS" : Bool;
         "New Cv" : DInt;
         pulses : DInt;
         "Reset timer" : Bool;
         F_trigger : Bool;
      END_STRUCT;
      "Leakage Control B" : Struct
         "Start Test" : Bool;
         "Start Test ONS" : Bool;
         "New Cv" : DInt;
         pulses : DInt;
         "Reset timer" : Bool;
         F_trigger : Bool;
      END_STRUCT;
      "Pump leakage" : Struct
         "A" : Bool;
         "B" : Bool;
      END_STRUCT;
   END_VAR
   VAR RETAIN
      "Volume Counter Enable button" : Bool;
   END_VAR
BEGIN
END_DATA_BLOCK

DATA_BLOCK "delaytimes"   // DB52
{ S7_Optimized_Access := 'TRUE' }
VERSION : 0.1
// stored: AutoNumber true, DBAccessibleFromOPCUA true, IsOnlyStoredInLoadMemory false, IsRetainMemResEnabled false, IsWriteProtectedInAS false, MemoryReserve 100
   VAR RETAIN
      "Outlet ON to pump ON A" : Int;
      "Outlet On to pump ON B" : Int;
   END_VAR
   VAR
      "Pump off to Inlet Close A" : Int;
      "Pump off to Inlet Close B" : Int;
   END_VAR
   VAR RETAIN
      "Pump off to Outlet Close" : Int;
      "Mixer ON to outlet ON" : Int;
      "outlet Off to mixer OFF" : Int;
      "Part Present On delay" : DInt;
      "Part Present Off Delay" : DInt;
      "Mixed flowrate error Delay time" : DInt := 2000;
   END_VAR
BEGIN
END_DATA_BLOCK

DATA_BLOCK "event For datalogging"   // DB216
{ S7_Optimized_Access := 'TRUE' }
VERSION : 0.1
// stored: AutoNumber false, DBAccessibleFromOPCUA true, IsOnlyStoredInLoadMemory false, IsRetainMemResEnabled false, IsWriteProtectedInAS false, MemoryReserve 100
   VAR
      "event number" : Int := 1;
      "event number Moved" : Int := 1;
      "trigger Datalogging on event change" : Bool := FALSE;
      "production completed" : String[25] := 'Production End';
      Metering_running : Bool;
      Function_String : Array[0..13] of String[25];
   END_VAR
BEGIN
   Function_String[1] := 'machine idle';
   Function_String[2] := 'metering program running';
   Function_String[3] := 'ratio Check running';
   Function_String[4] := 'metering shot running';
   Function_String[5] := 'metering cont. running';
   Function_String[6] := 'Pre run running';
   Function_String[7] := 'Flush running';
   Function_String[8] := 'Deaerate running';
   Function_String[9] := 'machine Faulty';
   Function_String[10] := 'emergency stop';
   Function_String[11] := 'regenration running';
   Function_String[12] := 'dosing completed';
END_DATA_BLOCK

DATA_BLOCK "level"   // DB72
{ S7_Optimized_Access := 'TRUE' }
VERSION : 0.1
// stored: AutoNumber true, DBAccessibleFromOPCUA true, IsOnlyStoredInLoadMemory false, IsRetainMemResEnabled false, IsWriteProtectedInAS false, MemoryReserve 100
   VAR RETAIN
      "A" : Struct
         "Low level" : Real := 20.0;
         "high level" : Real := 90.0;
         "level empty" : Real := 10.0;
      END_STRUCT;
      "B" : Struct
         "Low level" : Real := 20.0;
         "high level" : Real := 90.0;
         "level empty" : Real := 10.0;
      END_STRUCT;
      "present A1" : Real;
      "present A2" : Real;
      "present B1" : Real;
      "present B2" : Real;
   END_VAR
   VAR
      "Low level occured A1" : Bool;
      "Low level occured A2" : Bool;
      "High Level A" : Bool;
      "High Level B" : Bool;
      "Level Empty A2" : Bool;
      "Level Empty A1" : Bool;
      "Low level occured B1" : Bool;
      "Low level occured B2" : Bool;
      "Level Empty B1" : Bool;
      "Level Empty B2" : Bool;
      "Active vessel A" : Int;
      "Active vessel B" : Int;
      "scale A1" : Struct
         NormX : Real;
         scalx : Real;
      END_STRUCT;
      "scale B1" : Struct
         NormX : Real;
         scalx : Real;
      END_STRUCT;
      "Low level occured A" : Bool;
      "Low level occured B" : Bool;
      "Level Empty A" : Bool;
      "Level Empty B" : Bool;
      "Catridge low level A" : Bool;
      "Catridge low level B" : Bool;
      "Catridge level empty A" : Bool;
      "Catridge level empty B" : Bool;
      "Drum Level Low A1" : Bool;
      "Drum Level Low A2" : Bool;
      "Drum Level Empty A1" : Bool;
      "Drum Level Empty A2" : Bool;
      "Drum Level Low B1" : Bool;
      "Drum Level Low B2" : Bool;
      "Drum Level Empty B1" : Bool;
      "Drum Level Empty B2" : Bool;
   END_VAR
BEGIN
END_DATA_BLOCK

DATA_BLOCK "material Data Recipe"   // DB331
{ S7_Optimized_Access := 'TRUE' }
VERSION : 0.1
// stored: AutoNumber true, DBAccessibleFromOPCUA true, IsOnlyStoredInLoadMemory false, IsRetainMemResEnabled false, IsWriteProtectedInAS false, MemoryReserve 100
   VAR
      "Material 1" : Struct
         "Mixing ratio" : Real := 25.0;
         "Name A" : String[20] := 'resin1';
         "Name B" : String[20] := 'hardener1';
         "Density A" : Real;
         "Density B" : Real;
         "Viscosity A" : Real;
         "Vsicosity B" : Real;
         "A+" : String[21];
         "Name A+B" : String[42];
      END_STRUCT;
   END_VAR
   VAR RETAIN
      Selection : Int;
   END_VAR
   VAR
      "Selected material" : String;
   END_VAR
   VAR RETAIN
      "+symbol" : String := '+';
   END_VAR
BEGIN
END_DATA_BLOCK

DATA_BLOCK "mixer"   // DB74
{ S7_Optimized_Access := 'TRUE' }
VERSION : 0.1
// stored: AutoNumber true, DBAccessibleFromOPCUA true, IsOnlyStoredInLoadMemory false, IsRetainMemResEnabled false, IsWriteProtectedInAS false, MemoryReserve 100
   VAR RETAIN
      "mixer enable" : Int;
      "mixer control enable" : Int;
   END_VAR
   VAR
      "mixer enabled" : Bool;
      "mixer control enabled" : Bool;
   END_VAR
   VAR RETAIN
      "mixer speed at20 mA" : Real;
      "mixer Speed maximum" : Real;
      "mixer speed" : Real;
   END_VAR
   VAR
      "mixer control time" : Int;
   END_VAR
BEGIN
END_DATA_BLOCK

